C03633=1121.483,37.693,-52.816,179.793,7.035,149.366
C03634=1121.488,37.443,-52.800,179.792,7.030,149.365
C03635=1121.492,37.194,-52.785,179.791,7.026,149.364
C03636=1121.498,36.944,-52.770,179.790,7.022,149.364
C03637=1121.502,36.695,-52.755,179.789,7.018,149.363
C03638=1121.508,36.446,-52.739,179.788,7.014,149.363
C03639=1121.513,36.196,-52.723,179.787,7.010,149.362
C03640=1121.517,35.947,-52.708,179.786,7.006,149.361
C03641=1121.523,35.697,-52.693,179.785,7.002,149.361
C03642=1121.527,35.482,-52.680,179.784,6.997,149.360
C03643=1121.532,35.267,-52.667,179.783,6.994,149.360
C03644=1121.536,35.053,-52.653,179.782,6.991,149.359
C03645=1121.540,34.838,-52.641,179.781,6.987,149.359
C03646=1121.544,34.623,-52.627,179.780,6.983,149.358
C03647=1121.548,34.408,-52.614,179.779,6.979,149.358
C03648=1121.553,34.193,-52.601,179.778,6.976,149.357
C03649=1121.557,33.978,-52.588,179.777,6.973,149.356
C03650=1121.562,33.729,-52.573,179.776,6.968,149.356
C03651=1121.568,33.480,-52.557,179.775,6.964,149.355
C03652=1121.573,33.230,-52.542,179.774,6.960,149.355
C03653=1121.577,32.980,-52.527,179.773,6.955,149.354
C03654=1121.583,32.731,-52.511,179.772,6.951,149.353
C03655=1121.587,32.482,-52.496,179.771,6.947,149.353
C03656=1121.593,32.232,-52.481,179.770,6.942,149.352
C03657=1121.598,31.983,-52.466,179.769,6.938,149.351
C03658=1121.603,31.733,-52.451,179.768,6.934,149.351
C03659=1121.608,31.484,-52.436,179.767,6.929,149.350
C03660=1121.613,31.234,-52.421,179.766,6.925,149.349
C03661=1121.617,30.984,-52.405,179.765,6.921,149.349
C03662=1121.622,30.735,-52.390,179.764,6.916,149.348
C03663=1121.627,30.486,-52.375,179.762,6.912,149.347
C03664=1121.632,30.236,-52.361,179.761,6.908,149.347
C03665=1121.638,29.987,-52.345,179.760,6.904,149.346
C03666=1121.642,29.738,-52.330,179.759,6.899,149.345
C03667=1121.648,29.488,-52.315,179.758,6.895,149.345
C03668=1121.653,29.238,-52.300,179.757,6.891,149.344
C03669=1121.658,28.988,-52.285,179.756,6.886,149.343
C03670=1121.663,28.739,-52.270,179.755,6.882,149.343
C03671=1121.668,28.490,-52.255,179.754,6.878,149.342
C03672=1121.673,28.240,-52.240,179.753,6.873,149.341
C03673=1121.678,27.991,-52.225,179.752,6.869,149.341
C03674=1121.683,27.741,-52.211,179.751,6.864,149.340
C03675=1121.688,27.492,-52.196,179.750,6.860,149.339
C03676=1121.693,27.242,-52.181,179.749,6.856,149.339
C03677=1121.699,26.993,-52.166,179.748,6.851,149.338
C03678=1121.704,26.743,-52.151,179.747,6.847,149.337
C03679=1121.708,26.494,-52.136,179.746,6.843,149.337
C03680=1121.714,26.244,-52.122,179.745,6.838,149.336
C03681=1121.719,25.995,-52.107,179.744,6.834,149.335
C03682=1121.724,25.745,-52.092,179.743,6.829,149.335
C03683=1121.729,25.496,-52.077,179.742,6.825,149.334
C03684=1121.734,25.246,-52.062,179.741,6.821,149.333
C03685=1121.739,24.997,-52.047,179.740,6.816,149.333
C03686=1121.744,24.747,-52.033,179.739,6.812,149.332
C03687=1121.749,24.498,-52.018,179.739,6.807,149.331
C03688=1121.754,24.248,-52.003,179.738,6.803,149.330
C03689=1121.759,23.999,-51.988,179.736,6.799,149.330
C03690=1121.764,23.749,-51.973,179.735,6.794,149.329
C03691=1121.769,23.499,-51.959,179.734,6.790,149.328
C03692=1121.774,23.250,-51.944,179.734,6.785,149.328
C03693=1121.779,23.001,-51.930,179.733,6.781,149.327
C03694=1121.785,22.751,-51.915,179.732,6.777,149.326
C03695=1121.789,22.501,-51.900,179.731,6.772,149.326
C03696=1121.794,22.252,-51.886,179.730,6.768,149.325
C03697=1121.799,22.002,-51.871,179.729,6.763,149.324
C03698=1121.804,21.787,-51.858,179.729,6.760,149.323
C03699=1121.808,21.572,-51.846,179.728,6.756,149.323
C03700=1121.812,21.358,-51.833,179.727,6.752,149.322
C03701=1121.816,21.143,-51.821,179.726,6.749,149.322
C03702=1121.821,20.927,-51.808,179.725,6.745,149.321
C03703=1121.825,20.713,-51.796,179.725,6.741,149.320
C03704=1121.829,20.498,-51.783,179.724,6.737,149.320
C03705=1121.834,20.283,-51.770,179.723,6.733,149.319
C03706=1121.840,20.034,-51.756,179.722,6.729,149.318
C03707=1121.845,19.784,-51.742,179.721,6.725,149.318
C03708=1121.850,19.534,-51.728,179.721,6.720,149.317
C03709=1121.854,19.285,-51.713,179.720,6.716,149.316
C03710=1121.859,19.036,-51.698,179.719,6.711,149.316
C03711=1121.864,18.786,-51.684,179.717,6.706,149.315
C03712=1121.870,18.536,-51.669,179.716,6.701,149.314
C03713=1121.875,18.286,-51.655,179.715,6.697,149.313
C03714=1121.880,18.037,-51.641,179.715,6.692,149.313
C03715=1121.885,17.788,-51.626,179.714,6.688,149.312
C03716=1121.890,17.538,-51.612,179.713,6.683,149.311
C03717=1121.895,17.289,-51.597,179.712,6.679,149.310
C03718=1121.900,17.039,-51.583,179.711,6.675,149.310
C03719=1121.905,16.789,-51.569,179.711,6.670,149.309
C03720=1121.910,16.540,-51.555,179.709,6.666,149.308
C03721=1121.915,16.290,-51.541,179.709,6.661,149.307
C03722=1121.920,16.041,-51.526,179.708,6.657,149.307
C03723=1121.925,15.791,-51.512,179.707,6.652,149.306
C03724=1121.930,15.542,-51.497,179.706,6.648,149.305
C03725=1121.935,15.293,-51.483,179.706,6.643,149.304
C03726=1121.940,15.043,-51.469,179.705,6.639,149.304
C03727=1121.945,14.793,-51.455,179.704,6.634,149.303
C03728=1121.950,14.544,-51.440,179.703,6.630,149.302
C03729=1121.955,14.294,-51.426,179.703,6.625,149.301
C03730=1121.961,14.045,-51.412,179.702,6.621,149.301
C03731=1121.966,13.795,-51.398,179.700,6.615,149.300
C03732=1121.971,13.546,-51.384,179.699,6.611,149.299
C03733=1121.976,13.296,-51.369,179.699,6.606,149.298
C03734=1121.981,13.047,-51.355,179.698,6.602,149.297
C03735=1121.986,12.797,-51.341,179.697,6.597,149.297
C03736=1121.991,12.547,-51.327,179.697,6.592,149.296
C03737=1121.996,12.297,-51.313,179.696,6.588,149.295
C03738=1122.002,12.048,-51.299,179.695,6.583,149.294
C03739=1122.007,11.798,-51.285,179.694,6.579,149.294
C03740=1122.012,11.549,-51.271,179.693,6.574,149.293
C03741=1122.017,11.300,-51.257,179.693,6.569,149.292
C03742=1122.022,11.050,-51.243,179.692,6.565,149.291
C03743=1122.027,10.800,-51.228,179.691,6.560,149.290
C03744=1122.031,10.551,-51.215,179.690,6.555,149.290
C03745=1122.037,10.302,-51.201,179.689,6.551,149.289
C03746=1122.042,10.052,-51.187,179.689,6.546,149.288
C03747=1122.047,9.802,-51.173,179.688,6.542,149.287
C03748=1122.053,9.553,-51.159,179.687,6.537,149.286
C03749=1122.058,9.303,-51.145,179.686,6.532,149.285
C03750=1122.063,9.053,-51.131,179.686,6.527,149.285
C03751=1122.068,8.804,-51.118,179.685,6.523,149.284
C03752=1122.073,8.554,-51.104,179.684,6.518,149.283
C03753=1122.078,8.305,-51.089,179.684,6.514,149.282
C03754=1122.082,8.089,-51.078,179.683,6.509,149.281
C03755=1122.087,7.875,-51.066,179.682,6.506,149.281
C03756=1122.091,7.660,-51.053,179.682,6.502,149.280
C03757=1122.095,7.445,-51.042,179.681,6.498,149.279
C03758=1122.100,7.229,-51.030,179.681,6.494,149.278
C03759=1122.105,7.015,-51.017,179.681,6.490,149.278
C03760=1122.109,6.800,-51.006,179.681,6.487,149.277
C03761=1122.113,6.585,-50.994,179.680,6.482,149.276
C03762=1122.118,6.335,-50.980,179.680,6.477,149.275
C03763=1122.123,6.086,-50.967,179.679,6.474,149.275
C03764=1122.128,5.836,-50.953,179.679,6.469,149.274
C03765=1122.134,5.587,-50.939,179.678,6.464,149.273
C03766=1122.139,5.337,-50.925,179.678,6.459,149.272
C03767=1122.143,5.087,-50.912,179.677,6.455,149.271
C03768=1122.149,4.838,-50.898,179.677,6.451,149.270
C03769=1122.154,4.588,-50.884,179.677,6.446,149.269
C03770=1122.160,4.339,-50.870,179.676,6.442,149.269
C03771=1122.164,4.089,-50.857,179.675,6.437,149.268
C03772=1122.169,3.839,-50.843,179.674,6.432,149.267
C03773=1122.175,3.590,-50.829,179.674,6.428,149.266
C03774=1122.179,3.340,-50.816,179.674,6.424,149.265
C03775=1122.185,3.091,-50.802,179.673,6.419,149.264
C03776=1122.190,2.841,-50.789,179.672,6.415,149.264
C03777=1122.195,2.591,-50.774,179.672,6.410,149.263
C03778=1122.200,2.342,-50.761,179.671,6.405,149.262
C03779=1122.205,2.092,-50.748,179.671,6.400,149.261
C03780=1122.211,1.843,-50.734,179.670,6.397,149.260
C03781=1122.215,1.593,-50.721,179.670,6.392,149.259
C03782=1122.221,1.344,-50.707,179.669,6.387,149.259
C03783=1122.225,1.094,-50.694,179.669,6.383,149.258
C03784=1122.231,0.845,-50.680,179.668,6.378,149.257
C03785=1122.236,0.595,-50.666,179.667,6.374,149.256
C03786=1122.241,0.346,-50.653,179.667,6.370,149.255
C03787=1122.246,0.096,-50.639,179.667,6.365,149.254
C03788=1122.252,-0.153,-50.626,179.666,6.361,149.254
C03789=1122.256,-0.404,-50.613,179.665,6.356,149.253
C03790=1122.262,-0.653,-50.599,179.665,6.351,149.252
C03791=1122.266,-0.903,-50.586,179.664,6.346,149.251
C03792=1122.272,-1.152,-50.573,179.663,6.342,149.250
C03793=1122.276,-1.402,-50.559,179.663,6.338,149.249
C03794=1122.282,-1.651,-50.546,179.663,6.334,149.249
C03795=1122.287,-1.901,-50.531,179.662,6.329,149.248
C03796=1122.292,-2.150,-50.519,179.661,6.324,149.247
C03797=1122.298,-2.401,-50.505,179.661,6.320,149.246
C03798=1122.302,-2.649,-50.492,179.660,6.315,149.245
C03799=1122.308,-2.900,-50.478,179.659,6.311,149.245
C03800=1122.313,-3.149,-50.466,179.659,6.306,149.244
C03801=1122.318,-3.399,-50.451,179.658,6.301,149.243
C03802=1122.323,-3.648,-50.439,179.658,6.297,149.242
C03803=1122.328,-3.898,-50.425,179.657,6.293,149.241
C03804=1122.333,-4.147,-50.412,179.657,6.288,149.240
C03805=1122.338,-4.397,-50.398,179.656,6.284,149.240
C03806=1122.343,-4.647,-50.386,179.655,6.279,149.239
C03807=1122.349,-4.896,-50.373,179.655,6.274,149.238
C03808=1122.353,-5.146,-50.359,179.654,6.270,149.237
C03809=1122.359,-5.395,-50.346,179.653,6.265,149.236
C03810=1122.363,-5.611,-50.334,179.653,6.261,149.236
C03811=1122.368,-5.825,-50.323,179.653,6.258,149.235
C03812=1122.373,-6.041,-50.312,179.652,6.254,149.234
C03813=1122.377,-6.256,-50.300,179.652,6.250,149.234
C03814=1122.382,-6.471,-50.289,179.651,6.246,149.233
C03815=1122.385,-6.686,-50.278,179.650,6.242,149.232
C03816=1122.389,-6.901,-50.266,179.650,6.238,149.231
C03817=1122.394,-7.116,-50.255,179.649,6.234,149.231
C03818=1122.400,-7.367,-50.242,179.648,6.230,149.230
C03819=1122.404,-7.615,-50.229,179.648,6.225,149.229
C03820=1122.410,-7.865,-50.215,179.647,6.220,149.228
C03821=1122.415,-8.115,-50.202,179.646,6.216,149.228
C03822=1122.420,-8.364,-50.190,179.646,6.212,149.227
C03823=1122.426,-8.614,-50.177,179.646,6.207,149.226
C03824=1122.430,-8.864,-50.164,179.645,6.203,149.225
C03825=1122.435,-9.113,-50.151,179.644,6.198,149.224
C03826=1122.441,-9.362,-50.137,179.644,6.193,149.223
C03827=1122.445,-9.612,-50.124,179.643,6.189,149.222
C03828=1122.451,-9.861,-50.112,179.642,6.184,149.222
C03829=1122.456,-10.111,-50.098,179.642,6.179,149.221
C03830=1122.461,-10.361,-50.085,179.641,6.175,149.220
C03831=1122.466,-10.610,-50.073,179.640,6.170,149.219
C03832=1122.472,-10.860,-50.060,179.640,6.166,149.218
C03833=1122.476,-11.110,-50.047,179.639,6.161,149.218
C03834=1122.482,-11.359,-50.034,179.638,6.157,149.217
C03835=1122.487,-11.609,-50.021,179.638,6.152,149.216
C03836=1122.492,-11.859,-50.008,179.637,6.147,149.215
C03837=1122.497,-12.108,-49.995,179.636,6.143,149.214
C03838=1122.502,-12.358,-49.983,179.636,6.138,149.214
C03839=1122.507,-12.608,-49.969,179.635,6.133,149.213
C03840=1122.513,-12.857,-49.956,179.634,6.129,149.212
C03841=1122.518,-13.107,-49.944,179.634,6.124,149.211
C03842=1122.523,-13.356,-49.931,179.633,6.120,149.210
C03843=1122.528,-13.606,-49.918,179.632,6.115,149.210
C03844=1122.533,-13.856,-49.905,179.632,6.110,149.209
C03845=1122.538,-14.105,-49.892,179.631,6.106,149.208
C03846=1122.543,-14.355,-49.880,179.631,6.101,149.207
C03847=1122.549,-14.605,-49.866,179.630,6.097,149.206
C03848=1122.554,-14.854,-49.854,179.629,6.091,149.205
C03849=1122.559,-15.104,-49.842,179.628,6.086,149.204
C03850=1122.564,-15.354,-49.829,179.627,6.082,149.204
C03851=1122.569,-15.603,-49.816,179.627,6.077,149.203
C03852=1122.575,-15.853,-49.803,179.626,6.073,149.202
C03853=1122.580,-16.102,-49.790,179.625,6.068,149.201
C03854=1122.585,-16.351,-49.778,179.625,6.064,149.200
C03855=1122.590,-16.601,-49.765,179.624,6.059,149.200
C03856=1122.595,-16.851,-49.753,179.624,6.054,149.199
C03857=1122.600,-17.101,-49.740,179.623,6.050,149.198
C03858=1122.606,-17.350,-49.727,179.622,6.045,149.197
C03859=1122.611,-17.600,-49.715,179.622,6.040,149.196
C03860=1122.616,-17.850,-49.702,179.621,6.035,149.195
C03861=1122.621,-18.100,-49.690,179.620,6.030,149.195
C03862=1122.626,-18.349,-49.677,179.619,6.026,149.194
C03863=1122.631,-18.598,-49.665,179.619,6.021,149.193
C03864=1122.636,-18.848,-49.652,179.618,6.016,149.192
C03865=1122.641,-19.098,-49.640,179.617,6.012,149.191
C03866=1122.646,-19.313,-49.628,179.617,6.007,149.190
C03867=1122.651,-19.528,-49.618,179.617,6.004,149.190
C03868=1122.655,-19.744,-49.607,179.616,5.999,149.189
C03869=1122.660,-19.959,-49.597,179.615,5.996,149.188
C03870=1122.664,-20.174,-49.585,179.615,5.991,149.188
C03871=1122.668,-20.389,-49.575,179.614,5.987,149.187
C03872=1122.673,-20.605,-49.564,179.613,5.983,149.186
C03873=1122.677,-20.820,-49.554,179.612,5.979,149.186
C03874=1122.683,-21.069,-49.541,179.612,5.974,149.185
C03875=1122.688,-21.319,-49.528,179.612,5.969,149.184
C03876=1122.694,-21.568,-49.516,179.611,5.964,149.183
C03877=1122.699,-21.818,-49.504,179.610,5.959,149.182
C03878=1122.703,-22.068,-49.491,179.609,5.955,149.181
C03879=1122.709,-22.318,-49.479,179.609,5.950,149.180
C03880=1122.714,-22.567,-49.466,179.608,5.945,149.180
C03881=1122.719,-22.817,-49.455,179.608,5.940,149.179
C03882=1122.724,-23.066,-49.442,179.606,5.935,149.178
C03883=1122.730,-23.316,-49.430,179.606,5.930,149.177
C03884=1122.735,-23.566,-49.417,179.605,5.926,149.176
C03885=1122.739,-23.815,-49.405,179.605,5.921,149.175
C03886=1122.745,-24.065,-49.394,179.603,5.916,149.174
C03887=1122.750,-24.314,-49.381,179.603,5.911,149.174
C03888=1122.755,-24.564,-49.369,179.603,5.906,149.173
C03889=1122.760,-24.813,-49.356,179.602,5.901,149.172
C03890=1122.766,-25.063,-49.345,179.601,5.896,149.171
C03891=1122.771,-25.313,-49.333,179.601,5.891,149.170
C03892=1122.776,-25.562,-49.320,179.600,5.886,149.169
C03893=1122.781,-25.813,-49.308,179.598,5.881,149.168
C03894=1122.786,-26.062,-49.295,179.599,5.877,149.167
C03895=1122.792,-26.312,-49.283,179.600,5.872,149.166
C03896=1122.797,-26.561,-49.271,179.601,5.869,149.165
C03897=1122.802,-26.811,-49.259,179.602,5.865,149.164
C03898=1122.807,-27.060,-49.247,179.602,5.860,149.163
C03899=1122.812,-27.310,-49.235,179.603,5.857,149.162
C03900=1122.818,-27.560,-49.223,179.604,5.853,149.161
C03901=1122.823,-27.810,-49.211,179.604,5.848,149.160
C03902=1122.828,-28.060,-49.199,179.605,5.844,149.158
C03903=1122.833,-28.309,-49.186,179.605,5.840,149.158
C03904=1122.838,-28.559,-49.175,179.606,5.836,149.156
C03905=1122.843,-28.808,-49.163,179.607,5.832,149.155
C03906=1122.849,-29.058,-49.150,179.607,5.828,149.154
C03907=1122.854,-29.308,-49.138,179.607,5.823,149.153
C03908=1122.859,-29.558,-49.126,179.607,5.819,149.152
C03909=1122.865,-29.807,-49.114,179.607,5.815,149.151
C03910=1122.869,-30.057,-49.103,179.608,5.811,149.150
C03911=1122.874,-30.306,-49.090,179.608,5.807,149.149
C03912=1122.880,-30.556,-49.078,179.608,5.803,149.148
C03913=1122.885,-30.806,-49.066,179.609,5.799,149.147
C03914=1122.890,-31.055,-49.054,179.608,5.794,149.146
C03915=1122.895,-31.305,-49.042,179.608,5.790,149.146
C03916=1122.900,-31.555,-49.030,179.609,5.786,149.145
C03917=1122.906,-31.805,-49.019,179.608,5.781,149.144
C03918=1122.911,-32.054,-49.006,179.608,5.778,149.143
C03919=1122.916,-32.304,-48.994,179.608,5.773,149.142
C03920=1122.922,-32.553,-48.983,179.608,5.769,149.141
C03921=1122.927,-32.802,-48.971,179.607,5.764,149.140
C03922=1122.931,-33.018,-48.960,179.607,5.761,149.139
C03923=1122.936,-33.233,-48.950,179.607,5.757,149.139
C03924=1122.940,-33.448,-48.940,179.607,5.753,149.138
C03925=1122.945,-33.664,-48.929,179.606,5.749,149.137
C03926=1122.949,-33.879,-48.919,179.606,5.745,149.136
C03927=1122.954,-34.094,-48.909,179.606,5.741,149.136
C03928=1122.959,-34.309,-48.899,179.605,5.738,149.135
C03929=1122.962,-34.525,-48.888,179.605,5.733,149.134
C03930=1122.968,-34.775,-48.876,179.604,5.729,149.133
C03931=1122.973,-35.025,-48.865,179.604,5.724,149.132
C03932=1122.978,-35.273,-48.854,179.603,5.719,149.132
C03933=1122.984,-35.523,-48.842,179.602,5.715,149.131
C03934=1122.989,-35.773,-48.830,179.602,5.710,149.130
C03935=1122.994,-36.023,-48.817,179.601,5.706,149.129
C03936=1122.999,-36.272,-48.806,179.600,5.701,149.128
C03937=1123.005,-36.522,-48.794,179.599,5.695,149.128
C03938=1123.010,-36.772,-48.782,179.598,5.691,149.127
C03939=1123.015,-37.022,-48.771,179.598,5.686,149.126
C03940=1123.020,-37.272,-48.759,179.596,5.681,149.125
C03941=1123.025,-37.521,-48.748,179.596,5.676,149.124
C03942=1123.031,-37.771,-48.736,179.594,5.671,149.124
C03943=1123.036,-38.021,-48.724,179.594,5.666,149.123
C03944=1123.041,-38.270,-48.712,179.592,5.661,149.122
C03945=1123.046,-38.519,-48.700,179.592,5.656,149.121
C03946=1123.051,-38.769,-48.689,179.590,5.651,149.121
C03947=1123.057,-39.018,-48.678,179.589,5.646,149.120
C03948=1123.062,-39.268,-48.666,179.588,5.641,149.119
C03949=1123.067,-39.518,-48.654,179.587,5.636,149.118
C03950=1123.072,-39.768,-48.643,179.586,5.631,149.117
C03951=1123.078,-40.018,-48.631,179.584,5.626,149.117
C03952=1123.083,-40.267,-48.620,179.583,5.620,149.116
C03953=1123.089,-40.517,-48.609,179.582,5.615,149.115
C03954=1123.093,-40.767,-48.597,179.580,5.610,149.115
C03955=1123.099,-41.017,-48.585,179.579,5.603,149.114
C03956=1123.104,-41.266,-48.574,179.577,5.598,149.113
C03957=1123.110,-41.516,-48.563,179.576,5.593,149.112
C03958=1123.114,-41.765,-48.551,179.575,5.587,149.111
C03959=1123.120,-42.015,-48.539,179.572,5.581,149.111
C03960=1123.124,-42.265,-48.528,179.571,5.576,149.110
C03961=1123.130,-42.514,-48.517,179.569,5.570,149.109
C03962=1123.135,-42.764,-48.506,179.568,5.565,149.109
C03963=1123.141,-43.014,-48.494,179.566,5.559,149.108
C03964=1123.146,-43.263,-48.483,179.566,5.554,149.107
C03965=1123.151,-43.513,-48.472,179.566,5.549,149.106
C03966=1123.156,-43.763,-48.460,179.566,5.545,149.105
C03967=1123.161,-44.013,-48.450,179.566,5.540,149.104
C03968=1123.167,-44.262,-48.438,179.567,5.535,149.102
C03969=1123.172,-44.512,-48.427,179.566,5.530,149.101
C03970=1123.177,-44.762,-48.415,179.567,5.526,149.100
C03971=1123.183,-45.011,-48.405,179.567,5.521,149.099
C03972=1123.188,-45.261,-48.393,179.567,5.516,149.098
C03973=1123.193,-45.511,-48.381,179.567,5.512,149.097
C03974=1123.199,-45.760,-48.371,179.567,5.507,149.096
C03975=1123.203,-46.010,-48.360,179.568,5.502,149.095
C03976=1123.209,-46.260,-48.348,179.568,5.497,149.094
C03977=1123.214,-46.509,-48.337,179.567,5.492,149.093
C03978=1123.218,-46.725,-48.327,179.568,5.489,149.092
C03979=1123.223,-46.941,-48.318,179.568,5.485,149.091
C03980=1123.227,-47.156,-48.308,179.568,5.481,149.090
C03981=1123.232,-47.371,-48.299,179.569,5.476,149.089
C03982=1123.237,-47.587,-48.290,179.569,5.472,149.088
C03983=1123.242,-47.802,-48.279,179.569,5.468,149.087
C03984=1123.246,-48.017,-48.270,179.569,5.464,149.086
C03985=1123.251,-48.233,-48.260,179.569,5.460,149.085
C03986=1123.256,-48.482,-48.249,179.569,5.455,149.084
C03987=1123.260,-48.732,-48.238,179.569,5.451,149.083
C03988=1123.267,-48.982,-48.227,179.570,5.446,149.082
C03989=1123.271,-49.231,-48.216,179.570,5.441,149.081
C03990=1123.277,-49.481,-48.206,179.570,5.437,149.080
C03991=1123.282,-49.731,-48.194,179.570,5.432,149.079
C03992=1123.287,-49.981,-48.182,179.571,5.428,149.078
C03993=1123.293,-50.230,-48.172,179.571,5.423,149.077
C03994=1123.297,-50.480,-48.161,179.570,5.418,149.076
C03995=1123.304,-50.730,-48.150,179.571,5.413,149.075
C03996=1123.308,-50.979,-48.139,179.571,5.408,149.073
C03997=1123.313,-51.229,-48.128,179.571,5.404,149.072
C03998=1123.319,-51.478,-48.117,179.571,5.399,149.071
C03999=1123.324,-51.729,-48.106,179.572,5.395,149.070
C04000=1123.330,-51.978,-48.095,179.572,5.390,149.069
C04001=1123.334,-52.227,-48.084,179.572,5.385,149.068
C04002=1123.339,-52.478,-48.073,179.572,5.381,149.067
C04003=1123.345,-52.727,-48.062,179.572,5.376,149.066
C04004=1123.350,-52.977,-48.051,179.573,5.372,149.065
C04005=1123.356,-53.226,-48.040,179.573,5.366,149.064
C04006=1123.361,-53.476,-48.030,179.573,5.361,149.063
C04007=1123.367,-53.726,-48.018,179.573,5.357,149.062
C04008=1123.372,-53.976,-48.008,179.573,5.352,149.061
C04009=1123.377,-54.226,-47.997,179.574,5.348,149.059
C04010=1123.382,-54.475,-47.986,179.573,5.343,149.058
C04011=1123.387,-54.725,-47.976,179.574,5.339,149.057
C04012=1123.392,-54.974,-47.965,179.574,5.334,149.056
C04013=1123.398,-55.225,-47.953,179.574,5.329,149.055
C04014=1123.403,-55.474,-47.943,179.574,5.324,149.054
C04015=1123.408,-55.724,-47.932,179.575,5.319,149.053
C04016=1123.414,-55.973,-47.921,179.575,5.315,149.052
C04017=1123.419,-56.223,-47.910,179.575,5.310,149.051
C04018=1123.424,-56.473,-47.900,179.576,5.306,149.050
C04019=1123.430,-56.723,-47.888,179.575,5.301,149.049
C04020=1123.435,-56.973,-47.878,179.576,5.297,149.048
C04021=1123.440,-57.222,-47.867,179.576,5.292,149.047
C04022=1123.445,-57.472,-47.856,179.576,5.287,149.046
C04023=1123.450,-57.721,-47.846,179.576,5.282,149.044
C04024=1123.455,-57.971,-47.835,179.576,5.278,149.044
C04025=1123.461,-58.221,-47.825,179.577,5.273,149.042
C04026=1123.466,-58.471,-47.814,179.577,5.268,149.041
C04027=1123.471,-58.720,-47.803,179.577,5.264,149.040
C04028=1123.477,-58.970,-47.792,179.577,5.259,149.039
C04029=1123.482,-59.220,-47.782,179.577,5.254,149.038
C04030=1123.487,-59.470,-47.770,179.577,5.250,149.037
C04031=1123.493,-59.719,-47.760,179.577,5.245,149.036
C04032=1123.498,-59.969,-47.750,179.578,5.241,149.035
C04033=1123.503,-60.218,-47.739,179.578,5.236,149.034
C04034=1123.508,-60.434,-47.730,179.577,5.231,149.033
C04035=1123.513,-60.650,-47.721,179.576,5.227,149.032
C04036=1123.516,-60.865,-47.712,179.575,5.222,149.032
C04037=1123.521,-61.081,-47.703,179.575,5.218,149.031
C04038=1123.526,-61.296,-47.694,179.574,5.213,149.030
C04039=1123.530,-61.512,-47.684,179.573,5.209,149.029
C04040=1123.535,-61.727,-47.675,179.573,5.204,149.028
C04041=1123.539,-61.942,-47.666,179.572,5.200,149.028
C04042=1123.545,-62.192,-47.656,179.571,5.194,149.027
C04043=1123.550,-62.442,-47.646,179.571,5.189,149.026
C04044=1123.555,-62.691,-47.635,179.570,5.184,149.025
C04045=1123.560,-62.941,-47.624,179.569,5.179,149.024
C04046=1123.565,-63.191,-47.614,179.568,5.173,149.023
C04047=1123.571,-63.440,-47.604,179.567,5.168,149.022
C04048=1123.576,-63.690,-47.593,179.567,5.163,149.021
C04049=1123.582,-63.940,-47.583,179.566,5.157,149.020
C04050=1123.587,-64.190,-47.572,179.566,5.152,149.019
C04051=1123.592,-64.439,-47.561,179.565,5.147,149.018
C04052=1123.598,-64.689,-47.551,179.564,5.141,149.017
C04053=1123.603,-64.939,-47.541,179.564,5.136,149.016
C04054=1123.608,-65.189,-47.530,179.563,5.131,149.015
C04055=1123.614,-65.438,-47.520,179.563,5.126,149.014
C04056=1123.619,-65.688,-47.510,179.562,5.120,149.013
C04057=1123.624,-65.938,-47.499,179.562,5.115,149.013
C04058=1123.629,-66.187,-47.490,179.561,5.109,149.011
C04059=1123.634,-66.437,-47.479,179.561,5.105,149.011
C04060=1123.640,-66.687,-47.469,179.560,5.099,149.010
C04061=1123.645,-66.936,-47.459,179.560,5.094,149.008
C04062=1123.650,-67.187,-47.448,179.559,5.088,149.008
C04063=1123.656,-67.436,-47.438,179.558,5.084,149.007
C04064=1123.662,-67.686,-47.428,179.558,5.078,149.005
C04065=1123.666,-67.936,-47.418,179.558,5.073,149.005
C04066=1123.671,-68.185,-47.408,179.557,5.067,149.004
C04067=1123.677,-68.435,-47.397,179.557,5.062,149.002
C04068=1123.682,-68.685,-47.387,179.556,5.057,149.002
C04069=1123.688,-68.935,-47.377,179.556,5.052,149.000
C04070=1123.694,-69.185,-47.367,179.555,5.046,148.999
C04071=1123.698,-69.434,-47.357,179.555,5.041,148.998
C04072=1123.703,-69.684,-47.347,179.555,5.036,148.997
C04073=1123.709,-69.934,-47.337,179.554,5.030,148.996
C04074=1123.715,-70.183,-47.326,179.554,5.025,148.995
C04075=1123.719,-70.432,-47.317,179.553,5.019,148.994
C04076=1123.724,-70.683,-47.306,179.553,5.015,148.993
C04077=1123.730,-70.933,-47.297,179.553,5.009,148.992
C04078=1123.736,-71.182,-47.287,179.553,5.003,148.991
C04079=1123.741,-71.432,-47.277,179.552,4.999,148.990
C04080=1123.746,-71.682,-47.266,179.553,4.994,148.989
C04081=1123.751,-71.931,-47.256,179.552,4.988,148.988
C04082=1123.757,-72.182,-47.247,179.552,4.983,148.987
C04083=1123.762,-72.431,-47.237,179.552,4.978,148.986
C04084=1123.768,-72.680,-47.227,179.551,4.972,148.984
C04085=1123.773,-72.931,-47.216,179.551,4.967,148.984
C04086=1123.778,-73.181,-47.207,179.551,4.962,148.982
C04087=1123.784,-73.430,-47.197,179.551,4.956,148.981
C04088=1123.789,-73.680,-47.187,179.550,4.951,148.980
C04089=1123.795,-73.929,-47.177,179.551,4.946,148.979
C04090=1123.799,-74.145,-47.169,179.550,4.941,148.978
C04091=1123.804,-74.361,-47.160,179.550,4.937,148.977
C04092=1123.808,-74.576,-47.152,179.550,4.932,148.976
C04093=1123.813,-74.792,-47.143,179.550,4.927,148.975
C04094=1123.817,-75.007,-47.135,179.550,4.923,148.974
C04095=1123.822,-75.223,-47.126,179.550,4.918,148.973
C04096=1123.826,-75.439,-47.118,179.550,4.914,148.972
C04097=1123.832,-75.654,-47.109,179.550,4.910,148.971
C04098=1123.836,-75.904,-47.100,179.550,4.905,148.970
C04099=1123.842,-76.154,-47.090,179.550,4.899,148.969
C04100=1123.847,-76.403,-47.080,179.550,4.893,148.968
C04101=1123.853,-76.653,-47.071,179.550,4.888,148.967
C04102=1123.858,-76.903,-47.060,179.550,4.884,148.966
C04103=1123.863,-77.152,-47.051,179.550,4.878,148.965
C04104=1123.869,-77.402,-47.041,179.550,4.873,148.964
C04105=1123.874,-77.651,-47.032,179.550,4.868,148.962
C04106=1123.879,-77.902,-47.022,179.550,4.863,148.961
C04107=1123.885,-78.152,-47.012,179.550,4.857,148.960
C04108=1123.890,-78.401,-47.003,179.550,4.852,148.959
C04109=1123.896,-78.651,-46.992,179.550,4.847,148.958
C04110=1123.901,-78.901,-46.984,179.550,4.841,148.957
C04111=1123.906,-79.150,-46.973,179.550,4.836,148.955
C04112=1123.911,-79.400,-46.964,179.551,4.831,148.954
C04113=1123.917,-79.650,-46.954,179.551,4.826,148.953
C04114=1123.922,-79.900,-46.945,179.551,4.821,148.952
C04115=1123.928,-80.149,-46.935,179.551,4.816,148.951
C04116=1123.933,-80.399,-46.926,179.551,4.811,148.950
C04117=1123.938,-80.649,-46.916,179.551,4.805,148.948
C04118=1123.943,-80.899,-46.907,179.552,4.800,148.947
C04119=1123.949,-81.149,-46.897,179.552,4.795,148.946
C04120=1123.954,-81.399,-46.888,179.552,4.790,148.945
C04121=1123.959,-81.648,-46.877,179.552,4.785,148.944
C04122=1123.965,-81.898,-46.869,179.552,4.780,148.943
C04123=1123.970,-82.147,-46.858,179.552,4.774,148.941
C04124=1123.975,-82.397,-46.849,179.553,4.770,148.940
C04125=1123.981,-82.647,-46.840,179.553,4.765,148.939
C04126=1123.986,-82.897,-46.830,179.553,4.760,148.938
C04127=1123.992,-83.147,-46.821,179.554,4.755,148.937
C04128=1123.997,-83.396,-46.811,179.554,4.749,148.935
C04129=1124.002,-83.646,-46.802,179.555,4.744,148.934
C04130=1124.008,-83.896,-46.793,179.555,4.739,148.933
C04131=1124.013,-84.145,-46.783,179.555,4.734,148.932
C04132=1124.019,-84.396,-46.774,179.556,4.729,148.931
C04133=1124.024,-84.645,-46.765,179.556,4.724,148.929
C04134=1124.030,-84.895,-46.755,179.556,4.719,148.928
C04135=1124.035,-85.145,-46.746,179.556,4.714,148.927
C04136=1124.040,-85.395,-46.737,179.557,4.709,148.926
C04137=1124.045,-85.644,-46.727,179.558,4.704,148.924
C04138=1124.051,-85.894,-46.718,179.558,4.699,148.923
C04139=1124.056,-86.144,-46.709,179.558,4.693,148.922
C04140=1124.061,-86.393,-46.699,179.559,4.689,148.921
C04141=1124.067,-86.643,-46.690,179.559,4.684,148.920
C04142=1124.072,-86.893,-46.681,179.559,4.679,148.919
C04143=1124.077,-87.143,-46.671,179.560,4.674,148.917
C04144=1124.083,-87.392,-46.662,179.561,4.669,148.916
C04145=1124.088,-87.643,-46.652,179.561,4.664,148.915
C04146=1124.093,-87.858,-46.644,179.561,4.660,148.914
C04147=1124.097,-88.074,-46.637,179.562,4.655,148.913
C04148=1124.102,-88.289,-46.629,179.562,4.651,148.912
C04149=1124.107,-88.505,-46.620,179.563,4.647,148.911
C04150=1124.111,-88.721,-46.612,179.563,4.643,148.910
C04151=1124.116,-88.936,-46.604,179.564,4.639,148.908
C04152=1124.120,-89.151,-46.597,179.564,4.635,148.907
C04153=1124.125,-89.367,-46.589,179.565,4.630,148.906
C04154=1124.131,-89.617,-46.579,179.565,4.625,148.905
C04155=1124.136,-89.867,-46.570,179.565,4.620,148.904
C04156=1124.141,-90.117,-46.561,179.567,4.615,148.903
C04157=1124.147,-90.367,-46.551,179.567,4.610,148.901
C04158=1124.152,-90.617,-46.542,179.568,4.606,148.900
C04159=1124.157,-90.866,-46.534,179.568,4.601,148.899
C04160=1124.162,-91.116,-46.525,179.569,4.596,148.898
C04161=1124.169,-91.366,-46.516,179.570,4.592,148.896
C04162=1124.173,-91.615,-46.506,179.570,4.586,148.895
C04163=1124.179,-91.865,-46.497,179.571,4.582,148.894
C04164=1124.184,-92.115,-46.488,179.572,4.576,148.893
C04165=1124.190,-92.365,-46.479,179.572,4.572,148.891
C04166=1124.195,-92.615,-46.470,179.573,4.568,148.890
C04167=1124.200,-92.864,-46.461,179.573,4.563,148.889
C04168=1124.206,-93.115,-46.451,179.575,4.558,148.888
C04169=1124.211,-93.365,-46.442,179.575,4.553,148.886
C04170=1124.216,-93.614,-46.433,179.576,4.548,148.885
C04171=1124.222,-93.863,-46.424,179.576,4.544,148.884
C04172=1124.227,-94.113,-46.415,179.578,4.539,148.883
C04173=1124.233,-94.363,-46.406,179.578,4.534,148.881
C04174=1124.238,-94.613,-46.397,179.579,4.530,148.880
C04175=1124.243,-94.863,-46.388,179.579,4.525,148.879
C04176=1124.248,-95.112,-46.379,179.579,4.519,148.878
C04177=1124.254,-95.363,-46.370,179.579,4.514,148.877
C04178=1124.260,-95.612,-46.361,179.580,4.510,148.876
C04179=1124.265,-95.862,-46.352,179.580,4.505,148.875
C04180=1124.270,-96.111,-46.343,179.580,4.500,148.873
C04181=1124.275,-96.361,-46.335,179.580,4.495,148.872
C04182=1124.281,-96.611,-46.326,179.581,4.490,148.871
C04183=1124.286,-96.861,-46.316,179.581,4.485,148.870
C04184=1124.292,-97.111,-46.307,179.581,4.480,148.869
C04185=1124.297,-97.360,-46.299,179.582,4.475,148.867
C04186=1124.303,-97.610,-46.290,179.582,4.470,148.866
C04187=1124.308,-97.860,-46.281,179.583,4.465,148.865
C04188=1124.313,-98.110,-46.272,179.583,4.460,148.864
C04189=1124.318,-98.360,-46.263,179.583,4.455,148.863
C04190=1124.325,-98.609,-46.254,179.583,4.450,148.862
C04191=1124.330,-98.859,-46.245,179.583,4.445,148.861
C04192=1124.335,-99.109,-46.236,179.584,4.441,148.859
C04193=1124.340,-99.359,-46.227,179.584,4.436,148.858
C04194=1124.345,-99.609,-46.218,179.584,4.430,148.857
C04195=1124.351,-99.858,-46.210,179.584,4.425,148.856
C04196=1124.356,-100.108,-46.201,179.585,4.420,148.855
C04197=1124.361,-100.357,-46.192,179.585,4.415,148.853
C04198=1124.367,-100.608,-46.183,179.586,4.411,148.852
C04199=1124.373,-100.858,-46.174,179.586,4.405,148.851
C04200=1124.378,-101.107,-46.166,179.586,4.400,148.850
C04201=1124.384,-101.357,-46.157,179.586,4.395,148.849
C04202=1124.388,-101.573,-46.149,179.587,4.391,148.848
C04203=1124.393,-101.789,-46.142,179.586,4.386,148.847
C04204=1124.397,-102.004,-46.134,179.587,4.382,148.846
C04205=1124.402,-102.220,-46.126,179.587,4.378,148.845
C04206=1124.407,-102.436,-46.119,179.587,4.373,148.844
C04207=1124.411,-102.651,-46.112,179.588,4.369,148.843
C04208=1124.416,-102.867,-46.104,179.588,4.365,148.842
C04209=1124.421,-103.083,-46.097,179.588,4.360,148.841
C04210=1124.426,-103.332,-46.088,179.588,4.355,148.840
C04211=1124.431,-103.582,-46.079,179.588,4.350,148.838
C04212=1124.437,-103.832,-46.071,179.589,4.346,148.837
C04213=1124.442,-104.082,-46.062,179.589,4.341,148.836
C04214=1124.447,-104.332,-46.053,179.589,4.335,148.835
C04215=1124.453,-104.582,-46.044,179.590,4.330,148.834
C04216=1124.458,-104.831,-46.036,179.590,4.325,148.832
C04217=1124.464,-105.081,-46.028,179.590,4.320,148.831
C04218=1124.469,-105.331,-46.019,179.590,4.315,148.830
C04219=1124.475,-105.580,-46.010,179.590,4.310,148.829
C04220=1124.480,-105.830,-46.001,179.590,4.305,148.828
C04221=1124.485,-106.081,-45.993,179.590,4.300,148.827
C04222=1124.491,-106.330,-45.984,179.591,4.294,148.826
C04223=1124.496,-106.580,-45.976,179.591,4.289,148.824
C04224=1124.502,-106.830,-45.968,179.591,4.284,148.823
C04225=1124.506,-107.080,-45.959,179.591,4.279,148.822
C04226=1124.512,-107.329,-45.951,179.592,4.274,148.821
C04227=1124.517,-107.579,-45.943,179.592,4.269,148.820
C04228=1124.523,-107.829,-45.934,179.592,4.263,148.818
C04229=1124.528,-108.078,-45.925,179.592,4.258,148.817
C04230=1124.534,-108.329,-45.917,179.592,4.253,148.816
C04231=1124.539,-108.578,-45.908,179.592,4.248,148.815
C04232=1124.545,-108.828,-45.900,179.593,4.243,148.814
C04233=1124.550,-109.078,-45.891,179.593,4.238,148.813
C04234=1124.555,-109.328,-45.882,179.593,4.233,148.811
C04235=1124.560,-109.577,-45.875,179.593,4.228,148.810
C04236=1124.566,-109.827,-45.866,179.594,4.222,148.809
C04237=1124.572,-110.076,-45.858,179.594,4.217,148.808
C04238=1124.577,-110.327,-45.850,179.594,4.212,148.807
C04239=1124.582,-110.577,-45.841,179.594,4.207,148.805
C04240=1124.588,-110.826,-45.832,179.595,4.202,148.804
C04241=1124.594,-111.076,-45.824,179.595,4.196,148.803
C04242=1124.598,-111.326,-45.816,179.595,4.191,148.802
C04243=1124.604,-111.576,-45.808,179.595,4.186,148.801
C04244=1124.609,-111.826,-45.799,179.596,4.181,148.800
C04245=1124.615,-112.075,-45.791,179.596,4.176,148.798
C04246=1124.620,-112.325,-45.782,179.596,4.171,148.797
C04247=1124.625,-112.575,-45.775,179.596,4.166,148.796
C04248=1124.631,-112.824,-45.766,179.596,4.161,148.795
C04249=1124.636,-113.075,-45.758,179.596,4.155,148.794
C04250=1124.642,-113.324,-45.749,179.596,4.149,148.793
C04251=1124.648,-113.575,-45.741,179.596,4.144,148.791
C04252=1124.653,-113.823,-45.733,179.597,4.139,148.790
C04253=1124.658,-114.074,-45.725,179.597,4.134,148.789
C04254=1124.663,-114.324,-45.716,179.597,4.129,148.788
C04255=1124.669,-114.573,-45.708,179.597,4.124,148.787
C04256=1124.674,-114.824,-45.701,179.598,4.118,148.785
C04257=1124.680,-115.073,-45.692,179.598,4.113,148.784
C04258=1124.684,-115.289,-45.685,179.598,4.108,148.783
C04259=1124.690,-115.505,-45.678,179.598,4.103,148.782
C04260=1124.695,-115.721,-45.671,179.598,4.099,148.781
C04261=1124.698,-115.936,-45.664,179.598,4.095,148.780
C04262=1124.703,-116.152,-45.657,179.599,4.090,148.779
C04263=1124.708,-116.368,-45.650,179.599,4.085,148.778
C04264=1124.713,-116.584,-45.643,179.599,4.081,148.777
C04265=1124.717,-116.799,-45.636,179.599,4.076,148.776
C04266=1124.723,-117.049,-45.628,179.599,4.071,148.775
C04267=1124.729,-117.299,-45.620,179.600,4.066,148.773
C04268=1124.735,-117.549,-45.612,179.599,4.060,148.772
C04269=1124.739,-117.798,-45.604,179.600,4.055,148.771
C04270=1124.745,-118.048,-45.596,179.600,4.050,148.770
C04271=1124.751,-118.299,-45.588,179.600,4.044,148.769
C04272=1124.756,-118.548,-45.580,179.601,4.039,148.767
C04273=1124.761,-118.798,-45.572,179.600,4.033,148.766
C04274=1124.766,-119.047,-45.564,179.601,4.028,148.765
C04275=1124.772,-119.298,-45.556,179.601,4.023,148.764
C04276=1124.778,-119.547,-45.548,179.601,4.018,148.762
C04277=1124.782,-119.797,-45.540,179.601,4.012,148.761
C04278=1124.789,-120.047,-45.532,179.601,4.006,148.760
C04279=1124.794,-120.297,-45.524,179.601,4.001,148.759
C04280=1124.799,-120.546,-45.516,179.602,3.996,148.758
C04281=1124.804,-120.797,-45.508,179.601,3.990,148.756
C04282=1124.810,-121.046,-45.501,179.602,3.985,148.755
C04283=1124.816,-121.296,-45.493,179.602,3.980,148.754
C04284=1124.821,-121.546,-45.485,179.602,3.974,148.753
C04285=1124.826,-121.795,-45.477,179.602,3.969,148.752
C04286=1124.832,-122.046,-45.469,179.603,3.963,148.750
C04287=1124.837,-122.295,-45.461,179.603,3.958,148.749
C04288=1124.843,-122.546,-45.453,179.603,3.952,148.748
C04289=1124.848,-122.795,-45.446,179.603,3.947,148.747
C04290=1124.854,-123.045,-45.438,179.603,3.941,148.745
C04291=1124.859,-123.294,-45.430,179.603,3.935,148.744
C04292=1124.865,-123.544,-45.422,179.603,3.930,148.743
C04293=1124.869,-123.794,-45.414,179.604,3.925,148.742
C04294=1124.875,-124.044,-45.407,179.603,3.919,148.741
C04295=1124.881,-124.294,-45.399,179.604,3.914,148.739
C04296=1124.886,-124.544,-45.391,179.604,3.908,148.738
C04297=1124.892,-124.793,-45.384,179.604,3.902,148.737
C04298=1124.898,-125.043,-45.376,179.604,3.897,148.735
C04299=1124.902,-125.293,-45.369,179.604,3.891,148.734
C04300=1124.908,-125.543,-45.361,179.604,3.886,148.733
C04301=1124.913,-125.793,-45.353,179.605,3.881,148.732
C04302=1124.919,-126.043,-45.345,179.604,3.875,148.731
C04303=1124.925,-126.293,-45.338,179.605,3.869,148.729
C04304=1124.930,-126.543,-45.330,179.605,3.863,148.728
C04305=1124.935,-126.792,-45.323,179.605,3.858,148.727
C04306=1124.941,-127.042,-45.315,179.606,3.853,148.726
C04307=1124.946,-127.292,-45.307,179.605,3.847,148.724
C04308=1124.952,-127.542,-45.300,179.606,3.842,148.723
C04309=1124.958,-127.792,-45.292,179.606,3.835,148.722
C04310=1124.963,-128.041,-45.285,179.606,3.830,148.720
C04311=1124.968,-128.292,-45.277,179.606,3.824,148.719
C04312=1124.974,-128.541,-45.270,179.606,3.819,148.718
C04313=1124.980,-128.791,-45.262,179.606,3.813,148.717
C04314=1124.555,-128.781,-45.288,179.614,3.817,148.715
C04315=1124.551,-128.531,-45.295,179.614,3.823,148.716
C04316=1124.545,-128.282,-45.302,179.613,3.829,148.718
C04317=1124.539,-128.032,-45.310,179.613,3.834,148.719
C04318=1124.535,-127.782,-45.318,179.613,3.840,148.720
C04319=1124.529,-127.532,-45.326,179.613,3.845,148.722
C04320=1124.523,-127.283,-45.333,179.613,3.851,148.723
C04321=1124.518,-127.032,-45.341,179.612,3.857,148.724
C04322=1124.512,-126.783,-45.348,179.613,3.863,148.725
C04323=1124.506,-126.533,-45.356,179.612,3.868,148.727
C04324=1124.502,-126.283,-45.364,179.612,3.873,148.728
C04325=1124.496,-126.033,-45.372,179.612,3.879,148.729
C04326=1124.490,-125.783,-45.379,179.612,3.884,148.730
C04327=1124.485,-125.533,-45.387,179.612,3.891,148.732
C04328=1124.479,-125.284,-45.394,179.611,3.896,148.733
C04329=1124.475,-125.034,-45.402,179.611,3.901,148.734
C04330=1124.469,-124.784,-45.410,179.611,3.907,148.735
C04331=1124.463,-124.534,-45.418,179.611,3.912,148.737
C04332=1124.458,-124.284,-45.426,179.611,3.917,148.738
C04333=1124.452,-124.035,-45.433,179.611,3.923,148.739
C04334=1124.447,-123.784,-45.441,179.611,3.929,148.740
C04335=1124.441,-123.535,-45.449,179.610,3.934,148.742
C04336=1124.436,-123.285,-45.456,179.610,3.940,148.743
C04337=1124.431,-123.035,-45.465,179.610,3.945,148.744
C04338=1124.425,-122.786,-45.472,179.610,3.950,148.745
C04339=1124.420,-122.535,-45.480,179.610,3.956,148.747
C04340=1124.415,-122.286,-45.488,179.610,3.962,148.748
C04341=1124.408,-122.036,-45.495,179.609,3.967,148.749
C04342=1124.403,-121.786,-45.504,179.610,3.973,148.750
C04343=1124.398,-121.537,-45.512,179.609,3.978,148.751
C04344=1124.392,-121.286,-45.520,179.609,3.983,148.753
C04345=1124.387,-121.037,-45.527,179.608,3.989,148.754
C04346=1124.382,-120.786,-45.535,179.609,3.995,148.755
C04347=1124.376,-120.537,-45.544,179.608,4.000,148.756
C04348=1124.371,-120.287,-45.551,179.608,4.005,148.758
C04349=1124.365,-120.037,-45.559,179.608,4.011,148.759
C04350=1124.361,-119.788,-45.567,179.608,4.016,148.760
C04351=1124.355,-119.538,-45.575,179.608,4.021,148.761
C04352=1124.349,-119.288,-45.583,179.607,4.027,148.762
C04353=1124.344,-119.038,-45.591,179.607,4.032,148.764
C04354=1124.338,-118.789,-45.599,179.607,4.038,148.765
C04355=1124.333,-118.538,-45.607,179.607,4.043,148.766
C04356=1124.327,-118.289,-45.615,179.607,4.048,148.767
C04357=1124.322,-118.039,-45.623,179.607,4.053,148.768
C04358=1124.316,-117.789,-45.631,179.607,4.059,148.770
C04359=1124.311,-117.539,-45.639,179.607,4.064,148.771
C04360=1124.305,-117.290,-45.647,179.606,4.070,148.772
C04361=1124.300,-117.040,-45.656,179.606,4.075,148.773
C04362=1124.295,-116.790,-45.664,179.606,4.080,148.774
C04363=1124.290,-116.574,-45.671,179.606,4.085,148.776
C04364=1124.285,-116.359,-45.678,179.605,4.089,148.777
C04365=1124.281,-116.142,-45.685,179.606,4.094,148.778
C04366=1124.276,-115.926,-45.692,179.605,4.099,148.779
C04367=1124.271,-115.711,-45.699,179.605,4.103,148.780
C04368=1124.267,-115.495,-45.706,179.605,4.108,148.781
C04369=1124.262,-115.280,-45.713,179.605,4.112,148.782
C04370=1124.257,-115.064,-45.720,179.605,4.117,148.783
C04371=1124.252,-114.814,-45.729,179.604,4.122,148.784
C04372=1124.246,-114.565,-45.736,179.604,4.127,148.785
C04373=1124.241,-114.314,-45.744,179.604,4.133,148.786
C04374=1124.236,-114.064,-45.753,179.603,4.138,148.788
C04375=1124.230,-113.814,-45.761,179.604,4.144,148.789
C04376=1124.224,-113.565,-45.770,179.604,4.149,148.790
C04377=1124.219,-113.315,-45.777,179.603,4.154,148.791
C04378=1124.214,-113.065,-45.786,179.603,4.159,148.792
C04379=1124.208,-112.816,-45.794,179.603,4.164,148.794
C04380=1124.203,-112.566,-45.803,179.603,4.170,148.795
C04381=1124.198,-112.316,-45.812,179.603,4.174,148.796
C04382=1124.192,-112.066,-45.819,179.603,4.180,148.797
C04383=1124.187,-111.817,-45.828,179.602,4.185,148.798
C04384=1124.181,-111.567,-45.835,179.602,4.190,148.799
C04385=1124.176,-111.317,-45.844,179.602,4.195,148.801
C04386=1124.170,-111.066,-45.853,179.601,4.200,148.802
C04387=1124.165,-110.817,-45.861,179.601,4.205,148.803
C04388=1124.159,-110.567,-45.870,179.601,4.211,148.804
C04389=1124.155,-110.317,-45.878,179.601,4.216,148.805
C04390=1124.149,-110.068,-45.886,179.600,4.221,148.807
C04391=1124.143,-109.818,-45.894,179.600,4.226,148.808
C04392=1124.138,-109.568,-45.903,179.600,4.231,148.809
C04393=1124.133,-109.319,-45.912,179.600,4.237,148.810
C04394=1124.127,-109.068,-45.920,179.600,4.242,148.811
C04395=1124.122,-108.818,-45.929,179.600,4.248,148.813
C04396=1124.116,-108.569,-45.937,179.600,4.253,148.814
C04397=1124.111,-108.319,-45.946,179.599,4.258,148.815
C04398=1124.106,-108.069,-45.954,179.598,4.262,148.816
C04399=1124.100,-107.820,-45.962,179.599,4.267,148.817
C04400=1124.095,-107.570,-45.971,179.599,4.272,148.818
C04401=1124.090,-107.320,-45.979,179.598,4.277,148.820
C04402=1124.084,-107.071,-45.988,179.598,4.283,148.821
C04403=1124.079,-106.820,-45.996,179.598,4.288,148.822
C04404=1124.073,-106.570,-46.005,179.598,4.293,148.823
C04405=1124.068,-106.321,-46.014,179.597,4.298,148.824
C04406=1124.062,-106.071,-46.022,179.597,4.303,148.826
C04407=1124.057,-105.821,-46.031,179.597,4.308,148.827
C04408=1124.051,-105.572,-46.039,179.597,4.314,148.828
C04409=1124.046,-105.322,-46.048,179.596,4.319,148.829
C04410=1124.041,-105.072,-46.057,179.596,4.324,148.830
C04411=1124.035,-104.821,-46.065,179.596,4.329,148.831
C04412=1124.030,-104.572,-46.074,179.596,4.334,148.832
C04413=1124.024,-104.322,-46.083,179.596,4.339,148.834
C04414=1124.019,-104.073,-46.092,179.596,4.344,148.835
C04415=1124.014,-103.823,-46.100,179.595,4.349,148.836
C04416=1124.008,-103.573,-46.108,179.595,4.354,148.837
C04417=1124.003,-103.323,-46.117,179.594,4.359,148.838
C04418=1123.998,-103.073,-46.126,179.594,4.364,148.840
C04419=1123.993,-102.858,-46.134,179.594,4.369,148.841
C04420=1123.988,-102.642,-46.141,179.594,4.373,148.841
C04421=1123.984,-102.427,-46.149,179.593,4.377,148.843
C04422=1123.979,-102.211,-46.156,179.594,4.382,148.844
C04423=1123.974,-101.995,-46.163,179.593,4.386,148.845
C04424=1123.970,-101.779,-46.171,179.593,4.390,148.846
C04425=1123.965,-101.564,-46.179,179.593,4.395,148.847
C04426=1123.961,-101.348,-46.186,179.593,4.399,148.848
C04427=1123.956,-101.098,-46.195,179.592,4.404,148.849
C04428=1123.950,-100.848,-46.204,179.592,4.409,148.850
C04429=1123.944,-100.599,-46.213,179.592,4.414,148.851
C04430=1123.939,-100.349,-46.222,179.592,4.419,148.852
C04431=1123.934,-100.099,-46.231,179.591,4.424,148.853
C04432=1123.928,-99.849,-46.240,179.591,4.429,148.855
C04433=1123.923,-99.599,-46.249,179.591,4.434,148.856
C04434=1123.917,-99.350,-46.257,179.591,4.439,148.857
C04435=1123.912,-99.100,-46.266,179.590,4.444,148.858
C04436=1123.907,-98.850,-46.275,179.590,4.449,148.859
C04437=1123.901,-98.600,-46.285,179.589,4.454,148.861
C04438=1123.896,-98.350,-46.293,179.589,4.459,148.862
C04439=1123.890,-98.101,-46.302,179.589,4.464,148.863
C04440=1123.885,-97.851,-46.311,179.589,4.469,148.864
C04441=1123.880,-97.601,-46.320,179.588,4.473,148.865
C04442=1123.875,-97.352,-46.329,179.588,4.479,148.866
C04443=1123.869,-97.101,-46.338,179.588,4.484,148.867
C04444=1123.864,-96.852,-46.347,179.588,4.489,148.869
C04445=1123.858,-96.602,-46.356,179.588,4.494,148.870
C04446=1123.853,-96.353,-46.365,179.587,4.498,148.871
C04447=1123.848,-96.103,-46.373,179.587,4.504,148.872
C04448=1123.842,-95.853,-46.382,179.586,4.509,148.873
C04449=1123.837,-95.603,-46.392,179.586,4.514,148.874
C04450=1123.831,-95.353,-46.401,179.585,4.518,148.876
C04451=1123.826,-95.103,-46.410,179.585,4.524,148.877
C04452=1123.821,-94.853,-46.419,179.586,4.528,148.878
C04453=1123.815,-94.604,-46.428,179.585,4.533,148.879
C04454=1123.809,-94.354,-46.437,179.585,4.538,148.880
C04455=1123.804,-94.104,-46.445,179.583,4.543,148.882
C04456=1123.799,-93.855,-46.455,179.583,4.548,148.883
C04457=1123.793,-93.605,-46.465,179.582,4.552,148.884
C04458=1123.788,-93.355,-46.473,179.581,4.556,148.885
C04459=1123.783,-93.105,-46.482,179.581,4.562,148.887
C04460=1123.778,-92.855,-46.491,179.580,4.566,148.888
C04461=1123.772,-92.605,-46.501,179.580,4.572,148.889
C04462=1123.766,-92.356,-46.509,179.579,4.576,148.890
C04463=1123.761,-92.107,-46.519,179.578,4.581,148.892
C04464=1123.756,-91.857,-46.528,179.577,4.586,148.893
C04465=1123.750,-91.607,-46.537,179.577,4.590,148.894
C04466=1123.745,-91.357,-46.546,179.576,4.595,148.895
C04467=1123.740,-91.107,-46.555,179.575,4.600,148.897
C04468=1123.735,-90.858,-46.565,179.575,4.605,148.898
C04469=1123.729,-90.607,-46.574,179.574,4.610,148.899
C04470=1123.724,-90.358,-46.583,179.573,4.614,148.900
C04471=1123.719,-90.108,-46.592,179.573,4.619,148.902
C04472=1123.713,-89.858,-46.601,179.573,4.625,148.903
C04473=1123.708,-89.608,-46.611,179.572,4.629,148.904
C04474=1123.703,-89.358,-46.620,179.572,4.634,148.905
C04475=1123.697,-89.143,-46.628,179.571,4.638,148.906
C04476=1123.693,-88.927,-46.636,179.571,4.642,148.907
C04477=1123.689,-88.711,-46.644,179.570,4.647,148.908
C04478=1123.684,-88.496,-46.652,179.569,4.651,148.909
C04479=1123.679,-88.280,-46.660,179.569,4.655,148.910
C04480=1123.674,-88.065,-46.668,179.568,4.659,148.911
C04481=1123.670,-87.849,-46.676,179.568,4.663,148.913
C04482=1123.666,-87.634,-46.684,179.567,4.667,148.914
C04483=1123.660,-87.383,-46.693,179.567,4.673,148.915
C04484=1123.655,-87.134,-46.703,179.567,4.678,148.916
C04485=1123.650,-86.884,-46.712,179.566,4.682,148.917
C04486=1123.644,-86.634,-46.721,179.566,4.688,148.918
C04487=1123.639,-86.384,-46.730,179.565,4.693,148.920
C04488=1123.633,-86.135,-46.741,179.565,4.698,148.921
C04489=1123.628,-85.885,-46.749,179.564,4.702,148.922
C04490=1123.623,-85.635,-46.758,179.564,4.708,148.923
C04491=1123.617,-85.385,-46.769,179.564,4.713,148.925
C04492=1123.612,-85.136,-46.777,179.563,4.718,148.926
C04493=1123.607,-84.886,-46.788,179.563,4.723,148.927
C04494=1123.602,-84.636,-46.797,179.562,4.728,148.928
C04495=1123.596,-84.386,-46.805,179.562,4.733,148.929
C04496=1123.591,-84.137,-46.816,179.562,4.738,148.930
C04497=1123.586,-83.887,-46.825,179.562,4.743,148.932
C04498=1123.580,-83.637,-46.834,179.561,4.748,148.933
C04499=1123.575,-83.388,-46.844,179.560,4.753,148.934
C04500=1123.569,-83.137,-46.853,179.560,4.758,148.935
C04501=1123.564,-82.888,-46.863,179.560,4.763,148.937
C04502=1123.559,-82.638,-46.872,179.560,4.769,148.938
C04503=1123.553,-82.389,-46.882,179.560,4.774,148.939
C04504=1123.548,-82.139,-46.891,179.560,4.779,148.940
C04505=1123.542,-81.889,-46.900,179.559,4.784,148.941
C04506=1123.537,-81.640,-46.910,179.559,4.788,148.942
C04507=1123.531,-81.389,-46.919,179.559,4.794,148.944
C04508=1123.527,-81.140,-46.929,179.558,4.799,148.945
C04509=1123.521,-80.890,-46.938,179.558,4.804,148.946
C04510=1123.516,-80.640,-46.948,179.558,4.809,148.947
C04511=1123.511,-80.390,-46.958,179.558,4.814,148.948
C04512=1123.506,-80.141,-46.968,179.558,4.819,148.949
C04513=1123.500,-79.891,-46.977,179.558,4.825,148.951
C04514=1123.495,-79.641,-46.987,179.557,4.830,148.952
C04515=1123.489,-79.391,-46.996,179.557,4.835,148.953
C04516=1123.483,-79.142,-47.006,179.557,4.840,148.954
C04517=1123.479,-78.892,-47.016,179.557,4.845,148.955
C04518=1123.473,-78.642,-47.025,179.557,4.850,148.956
C04519=1123.468,-78.393,-47.035,179.557,4.855,148.958
C04520=1123.462,-78.143,-47.045,179.557,4.861,148.959
C04521=1123.458,-77.893,-47.055,179.557,4.867,148.960
C04522=1123.452,-77.643,-47.064,179.557,4.872,148.961
C04523=1123.446,-77.393,-47.074,179.557,4.877,148.962
C04524=1123.441,-77.144,-47.084,179.556,4.882,148.963
C04525=1123.435,-76.894,-47.093,179.556,4.887,148.965
C04526=1123.430,-76.644,-47.104,179.556,4.892,148.966
C04527=1123.425,-76.395,-47.113,179.556,4.897,148.967
C04528=1123.420,-76.144,-47.123,179.557,4.903,148.968
C04529=1123.415,-75.895,-47.133,179.557,4.908,148.969
C04530=1123.409,-75.645,-47.142,179.557,4.913,148.970
C04531=1123.404,-75.429,-47.151,179.557,4.918,148.971
C04532=1123.399,-75.214,-47.159,179.557,4.922,148.972
C04533=1123.395,-74.999,-47.168,179.557,4.927,148.973
C04534=1123.390,-74.783,-47.176,179.556,4.931,148.974
C04535=1123.386,-74.567,-47.186,179.557,4.936,148.975
C04536=1123.381,-74.352,-47.193,179.557,4.941,148.976
C04537=1123.376,-74.137,-47.202,179.557,4.945,148.977
C04538=1123.372,-73.921,-47.210,179.557,4.950,148.978
C04539=1123.367,-73.671,-47.221,179.557,4.955,148.979
C04540=1123.361,-73.421,-47.230,179.557,4.961,148.980
C04541=1123.356,-73.172,-47.240,179.558,4.965,148.981
C04542=1123.351,-72.922,-47.250,179.558,4.971,148.982
C04543=1123.345,-72.672,-47.261,179.558,4.976,148.983
C04544=1123.340,-72.423,-47.270,179.559,4.981,148.984
C04545=1123.334,-72.173,-47.280,179.558,4.987,148.986
C04546=1123.329,-71.923,-47.290,179.558,4.992,148.987
C04547=1123.324,-71.673,-47.300,179.559,4.997,148.988
C04548=1123.319,-71.424,-47.310,179.559,5.002,148.989
C04549=1123.313,-71.174,-47.320,179.559,5.008,148.990
C04550=1123.308,-70.923,-47.330,179.560,5.013,148.991
C04551=1123.302,-70.674,-47.340,179.560,5.018,148.992
C04552=1123.297,-70.424,-47.351,179.560,5.023,148.993
C04553=1123.292,-70.175,-47.360,179.561,5.029,148.994
C04554=1123.287,-69.925,-47.371,179.561,5.034,148.995
C04555=1123.281,-69.675,-47.381,179.561,5.040,148.996
C04556=1123.276,-69.426,-47.391,179.562,5.044,148.997
C04557=1123.270,-69.176,-47.401,179.562,5.050,148.998
C04558=1123.266,-68.926,-47.411,179.563,5.055,148.999
C04559=1123.260,-68.677,-47.422,179.562,5.060,149.000
C04560=1123.254,-68.427,-47.431,179.563,5.066,149.001
C04561=1123.249,-68.176,-47.442,179.563,5.071,149.002
C04562=1123.244,-67.927,-47.452,179.564,5.077,149.003
C04563=1123.238,-67.677,-47.462,179.564,5.082,149.004
C04564=1123.234,-67.427,-47.472,179.565,5.087,149.005
C04565=1123.228,-67.178,-47.482,179.565,5.092,149.006
C04566=1123.223,-66.928,-47.492,179.565,5.097,149.007
C04567=1123.218,-66.678,-47.503,179.566,5.103,149.008
C04568=1123.212,-66.428,-47.513,179.567,5.108,149.009
C04569=1123.207,-66.179,-47.523,179.567,5.114,149.010
C04570=1123.202,-65.929,-47.535,179.568,5.118,149.011
C04571=1123.196,-65.680,-47.545,179.569,5.124,149.012
C04572=1123.191,-65.430,-47.555,179.568,5.129,149.013
C04573=1123.186,-65.180,-47.565,179.569,5.135,149.014
C04574=1123.181,-64.931,-47.575,179.570,5.140,149.015
C04575=1123.175,-64.681,-47.586,179.571,5.145,149.016
C04576=1123.170,-64.431,-47.596,179.572,5.151,149.017
C04577=1123.165,-64.181,-47.606,179.572,5.156,149.018
C04578=1123.160,-63.931,-47.617,179.573,5.161,149.019
C04579=1123.154,-63.682,-47.627,179.573,5.166,149.020
C04580=1123.149,-63.433,-47.638,179.574,5.172,149.021
C04581=1123.144,-63.182,-47.649,179.575,5.177,149.022
C04582=1123.138,-62.933,-47.659,179.575,5.182,149.023
C04583=1123.133,-62.683,-47.669,179.576,5.187,149.024
C04584=1123.128,-62.433,-47.680,179.577,5.192,149.025
C04585=1123.123,-62.183,-47.691,179.578,5.198,149.026
C04586=1123.117,-61.934,-47.701,179.579,5.203,149.026
C04587=1123.113,-61.718,-47.710,179.579,5.208,149.027
C04588=1123.108,-61.503,-47.720,179.580,5.212,149.028
C04589=1123.103,-61.287,-47.729,179.580,5.217,149.029
C04590=1123.099,-61.072,-47.738,179.581,5.222,149.030
C04591=1123.095,-60.857,-47.747,179.582,5.226,149.030
C04592=1123.090,-60.641,-47.756,179.583,5.231,149.031
C04593=1123.086,-60.426,-47.766,179.583,5.235,149.032
C04594=1123.081,-60.210,-47.775,179.584,5.240,149.033
C04595=1123.075,-59.961,-47.785,179.584,5.244,149.034
C04596=1123.070,-59.711,-47.796,179.583,5.249,149.035
C04597=1123.065,-59.462,-47.807,179.583,5.253,149.036
C04598=1123.060,-59.211,-47.817,179.583,5.258,149.037
C04599=1123.054,-58.962,-47.827,179.583,5.263,149.038
C04600=1123.050,-58.712,-47.839,179.583,5.267,149.039
C04601=1123.044,-58.463,-47.849,179.583,5.272,149.040
C04602=1123.039,-58.212,-47.859,179.582,5.277,149.041
C04603=1123.033,-57.963,-47.871,179.582,5.281,149.042
C04604=1123.028,-57.713,-47.881,179.582,5.286,149.043
C04605=1123.022,-57.463,-47.892,179.582,5.291,149.044
C04606=1123.018,-57.214,-47.903,179.581,5.295,149.046
C04607=1123.012,-56.964,-47.913,179.581,5.300,149.047
C04608=1123.008,-56.715,-47.924,179.582,5.305,149.048
C04609=1123.002,-56.465,-47.935,179.581,5.309,149.049
C04610=1122.996,-56.214,-47.946,179.581,5.314,149.050
C04611=1122.991,-55.965,-47.957,179.581,5.318,149.051
C04612=1122.986,-55.715,-47.967,179.581,5.323,149.052
C04613=1122.981,-55.466,-47.979,179.580,5.328,149.053
C04614=1122.976,-55.216,-47.989,179.580,5.332,149.054
C04615=1122.971,-54.967,-48.000,179.580,5.338,149.055
C04616=1122.965,-54.717,-48.011,179.580,5.342,149.056
C04617=1122.960,-54.467,-48.022,179.580,5.347,149.057
C04618=1122.955,-54.217,-48.033,179.579,5.351,149.058
C04619=1122.950,-53.968,-48.044,179.579,5.356,149.060
C04620=1122.945,-53.718,-48.054,179.579,5.360,149.060
C04621=1122.939,-53.468,-48.066,179.579,5.365,149.062
C04622=1122.934,-53.218,-48.076,179.579,5.370,149.063
C04623=1122.928,-52.969,-48.087,179.579,5.374,149.064
C04624=1122.923,-52.719,-48.098,179.579,5.380,149.065
C04625=1122.918,-52.469,-48.110,179.578,5.384,149.066
C04626=1122.912,-52.219,-48.120,179.578,5.389,149.067
C04627=1122.908,-51.970,-48.131,179.578,5.393,149.068
C04628=1122.902,-51.720,-48.141,179.578,5.398,149.069
C04629=1122.897,-51.470,-48.153,179.578,5.403,149.070
C04630=1122.892,-51.221,-48.165,179.577,5.407,149.071
C04631=1122.886,-50.971,-48.175,179.577,5.412,149.072
C04632=1122.881,-50.721,-48.187,179.577,5.417,149.074
C04633=1122.875,-50.472,-48.197,179.577,5.421,149.074
C04634=1122.871,-50.222,-48.208,179.577,5.427,149.076
C04635=1122.866,-49.972,-48.219,179.576,5.431,149.077
C04636=1122.859,-49.723,-48.230,179.577,5.436,149.078
C04637=1122.855,-49.473,-48.242,179.576,5.440,149.079
C04638=1122.850,-49.223,-48.252,179.576,5.445,149.080
C04639=1122.844,-48.974,-48.264,179.575,5.449,149.081
C04640=1122.839,-48.724,-48.275,179.576,5.454,149.082
C04641=1122.834,-48.474,-48.286,179.576,5.459,149.083
C04642=1122.828,-48.224,-48.297,179.575,5.464,149.084
C04643=1122.823,-48.009,-48.306,179.575,5.468,149.085
C04644=1122.819,-47.794,-48.316,179.575,5.472,149.086
C04645=1122.814,-47.579,-48.326,179.574,5.476,149.087
C04646=1122.810,-47.363,-48.335,179.575,5.480,149.088
C04647=1122.806,-47.148,-48.345,179.575,5.484,149.089
C04648=1122.801,-46.932,-48.355,179.574,5.488,149.090
C04649=1122.797,-46.717,-48.364,179.574,5.492,149.091
C04650=1122.792,-46.502,-48.374,179.574,5.496,149.092
C04651=1122.787,-46.252,-48.386,179.574,5.501,149.093
C04652=1122.781,-46.002,-48.396,179.573,5.506,149.094
C04653=1122.777,-45.753,-48.407,179.574,5.510,149.095
C04654=1122.771,-45.503,-48.419,179.573,5.515,149.096
C04655=1122.766,-45.254,-48.430,179.573,5.520,149.097
C04656=1122.760,-45.003,-48.441,179.573,5.525,149.098
C04657=1122.756,-44.753,-48.453,179.573,5.529,149.099
C04658=1122.750,-44.505,-48.464,179.573,5.534,149.100
C04659=1122.745,-44.255,-48.475,179.572,5.538,149.101
C04660=1122.740,-44.004,-48.486,179.572,5.544,149.103
C04661=1122.734,-43.754,-48.498,179.572,5.547,149.103
C04662=1122.729,-43.506,-48.509,179.572,5.553,149.105
C04663=1122.724,-43.256,-48.521,179.572,5.558,149.106
C04664=1122.719,-43.006,-48.532,179.572,5.563,149.107
C04665=1122.713,-42.756,-48.543,179.573,5.568,149.108
C04666=1122.708,-42.506,-48.554,179.575,5.574,149.108
C04667=1122.703,-42.257,-48.565,179.577,5.579,149.109
C04668=1122.698,-42.007,-48.577,179.579,5.586,149.110
C04669=1122.693,-41.758,-48.588,179.580,5.591,149.110
C04670=1122.687,-41.508,-48.600,179.582,5.596,149.111
C04671=1122.682,-41.258,-48.611,179.583,5.602,149.112
C04672=1122.677,-41.009,-48.623,179.585,5.607,149.113
C04673=1122.672,-40.759,-48.635,179.586,5.613,149.114
C04674=1122.666,-40.510,-48.646,179.587,5.618,149.114
C04675=1122.661,-40.260,-48.658,179.589,5.623,149.115
C04676=1122.656,-40.010,-48.669,179.590,5.629,149.116
C04677=1122.651,-39.760,-48.681,179.591,5.634,149.116
C04678=1122.646,-39.511,-48.692,179.593,5.639,149.117
C04679=1122.640,-39.261,-48.704,179.594,5.645,149.118
C04680=1122.635,-39.011,-48.716,179.595,5.649,149.119
C04681=1122.630,-38.762,-48.727,179.596,5.655,149.120
C04682=1122.624,-38.512,-48.739,179.598,5.660,149.120
C04683=1122.620,-38.262,-48.750,179.598,5.664,149.121
C04684=1122.614,-38.012,-48.762,179.600,5.670,149.122
C04685=1122.608,-37.763,-48.774,179.600,5.674,149.123
C04686=1122.604,-37.513,-48.785,179.602,5.680,149.123
C04687=1122.598,-37.263,-48.797,179.602,5.684,149.124
C04688=1122.593,-37.013,-48.809,179.603,5.689,149.125
C04689=1122.588,-36.764,-48.820,179.604,5.694,149.126
C04690=1122.583,-36.515,-48.833,179.605,5.699,149.127
C04691=1122.577,-36.265,-48.844,179.606,5.704,149.127
C04692=1122.572,-36.015,-48.856,179.606,5.709,149.128
C04693=1122.567,-35.765,-48.868,179.607,5.713,149.129
C04694=1122.561,-35.516,-48.879,179.608,5.718,149.130
C04695=1122.556,-35.266,-48.891,179.608,5.723,149.131
C04696=1122.552,-35.017,-48.903,179.609,5.727,149.131
C04697=1122.546,-34.767,-48.915,179.610,5.732,149.132
C04698=1122.541,-34.517,-48.927,179.610,5.736,149.133
C04699=1122.536,-34.302,-48.937,179.610,5.740,149.134
C04700=1122.532,-34.086,-48.948,179.611,5.744,149.135
C04701=1122.527,-33.871,-48.958,179.612,5.748,149.135
C04702=1122.523,-33.657,-48.968,179.612,5.752,149.136
C04703=1122.518,-33.440,-48.978,179.612,5.755,149.137
C04704=1122.514,-33.225,-48.988,179.613,5.760,149.138
C04705=1122.509,-33.010,-48.999,179.613,5.764,149.138
C04706=1122.505,-32.795,-49.009,179.613,5.767,149.139
C04707=1122.499,-32.545,-49.021,179.613,5.771,149.140
C04708=1122.494,-32.296,-49.033,179.613,5.776,149.141
C04709=1122.489,-32.046,-49.044,179.614,5.781,149.142
C04710=1122.484,-31.796,-49.056,179.614,5.785,149.143
C04711=1122.479,-31.547,-49.069,179.614,5.789,149.144
C04712=1122.473,-31.297,-49.081,179.614,5.793,149.145
C04713=1122.468,-31.047,-49.093,179.614,5.797,149.145
C04714=1122.464,-30.798,-49.105,179.613,5.802,149.147
C04715=1122.458,-30.548,-49.117,179.614,5.806,149.148
C04716=1122.453,-30.298,-49.129,179.614,5.810,149.148
C04717=1122.448,-30.049,-49.141,179.613,5.814,149.149
C04718=1122.442,-29.799,-49.153,179.613,5.819,149.150
C04719=1122.437,-29.550,-49.166,179.613,5.823,149.151
C04720=1122.432,-29.300,-49.177,179.612,5.826,149.152
C04721=1122.427,-29.050,-49.189,179.612,5.831,149.153
C04722=1122.422,-28.801,-49.201,179.612,5.835,149.154
C04723=1122.416,-28.551,-49.213,179.611,5.839,149.155
C04724=1122.411,-28.301,-49.226,179.610,5.843,149.157
C04725=1122.406,-28.052,-49.238,179.610,5.847,149.157
C04726=1122.400,-27.802,-49.250,179.610,5.852,149.159
C04727=1122.396,-27.553,-49.262,179.609,5.856,149.160
C04728=1122.391,-27.303,-49.274,179.609,5.860,149.161
C04729=1122.385,-27.053,-49.286,179.608,5.864,149.162
C04730=1122.380,-26.803,-49.298,179.607,5.868,149.163
C04731=1122.375,-26.553,-49.311,179.606,5.872,149.164
C04732=1122.370,-26.303,-49.323,179.605,5.876,149.165
C04733=1122.365,-26.054,-49.335,179.605,5.880,149.166
C04734=1122.359,-25.804,-49.347,179.605,5.885,149.167
C04735=1122.354,-25.555,-49.360,179.606,5.890,149.168
C04736=1122.350,-25.305,-49.371,179.606,5.894,149.169
C04737=1122.345,-25.056,-49.384,179.607,5.899,149.170
C04738=1122.339,-24.806,-49.396,179.608,5.905,149.171
C04739=1122.334,-24.557,-49.408,179.608,5.909,149.172
C04740=1122.329,-24.307,-49.420,179.609,5.914,149.173
C04741=1122.323,-24.057,-49.433,179.609,5.919,149.173
C04742=1122.318,-23.807,-49.445,179.610,5.924,149.174
C04743=1122.313,-23.558,-49.457,179.611,5.929,149.175
C04744=1122.307,-23.308,-49.469,179.612,5.933,149.176
C04745=1122.302,-23.059,-49.482,179.612,5.938,149.177
C04746=1122.297,-22.809,-49.494,179.613,5.944,149.178
C04747=1122.292,-22.559,-49.507,179.614,5.948,149.179
C04748=1122.287,-22.310,-49.519,179.614,5.953,149.180
C04749=1122.282,-22.060,-49.531,179.615,5.957,149.180
C04750=1122.277,-21.810,-49.544,179.616,5.962,149.181
C04751=1122.271,-21.560,-49.556,179.617,5.968,149.182
C04752=1122.266,-21.311,-49.568,179.617,5.972,149.183
C04753=1122.261,-21.062,-49.581,179.618,5.977,149.184
C04754=1122.256,-20.812,-49.593,179.618,5.982,149.185
C04755=1122.251,-20.597,-49.604,179.619,5.986,149.185
C04756=1122.246,-20.381,-49.615,179.619,5.990,149.186
C04757=1122.243,-20.166,-49.625,179.620,5.994,149.187
C04758=1122.238,-19.951,-49.637,179.621,5.999,149.188
C04759=1122.233,-19.736,-49.647,179.621,6.002,149.188
C04760=1122.229,-19.521,-49.658,179.622,6.007,149.189
C04761=1122.224,-19.306,-49.669,179.623,6.010,149.190
C04762=1122.220,-19.090,-49.680,179.623,6.015,149.190
C04763=1122.215,-18.841,-49.693,179.624,6.019,149.191
C04764=1122.209,-18.591,-49.704,179.624,6.024,149.192
C04765=1122.204,-18.342,-49.717,179.625,6.029,149.193
C04766=1122.200,-18.092,-49.730,179.625,6.034,149.194
C04767=1122.194,-17.842,-49.743,179.626,6.038,149.194
C04768=1122.189,-17.593,-49.755,179.628,6.043,149.195
C04769=1122.184,-17.343,-49.767,179.628,6.048,149.196
C04770=1122.178,-17.093,-49.780,179.629,6.053,149.197
C04771=1122.174,-16.843,-49.793,179.629,6.057,149.198
C04772=1122.168,-16.594,-49.806,179.630,6.062,149.199
C04773=1122.163,-16.345,-49.818,179.630,6.067,149.200
C04774=1122.158,-16.095,-49.831,179.631,6.071,149.200
C04775=1122.153,-15.845,-49.843,179.632,6.076,149.201
C04776=1122.147,-15.595,-49.856,179.632,6.081,149.202
C04777=1122.142,-15.346,-49.869,179.633,6.085,149.203
C04778=1122.137,-15.096,-49.882,179.634,6.090,149.204
C04779=1122.132,-14.847,-49.894,179.634,6.094,149.204
C04780=1122.127,-14.597,-49.908,179.635,6.099,149.205
C04781=1122.122,-14.347,-49.920,179.635,6.104,149.206
C04782=1122.117,-14.098,-49.933,179.636,6.108,149.207
C04783=1122.111,-13.849,-49.946,179.637,6.114,149.208
C04784=1122.107,-13.599,-49.959,179.638,6.118,149.209
C04785=1122.101,-13.349,-49.972,179.639,6.123,149.209
C04786=1122.096,-13.100,-49.984,179.639,6.128,149.210
C04787=1122.091,-12.850,-49.997,179.640,6.132,149.211
C04788=1122.086,-12.600,-50.011,179.641,6.137,149.212
C04789=1122.080,-12.351,-50.023,179.641,6.141,149.213
C04790=1122.076,-12.101,-50.036,179.642,6.146,149.214
C04791=1122.071,-11.852,-50.049,179.642,6.151,149.214
C04792=1122.065,-11.602,-50.062,179.643,6.155,149.215
C04793=1122.060,-11.353,-50.075,179.644,6.160,149.216
C04794=1122.055,-11.103,-50.087,179.644,6.165,149.217
C04795=1122.049,-10.853,-50.101,179.645,6.169,149.218
C04796=1122.044,-10.604,-50.113,179.646,6.174,149.218
C04797=1122.040,-10.354,-50.126,179.646,6.178,149.219
C04798=1122.034,-10.104,-50.139,179.647,6.183,149.220
C04799=1122.029,-9.854,-50.152,179.648,6.187,149.221
C04800=1122.024,-9.605,-50.165,179.648,6.192,149.222
C04801=1122.018,-9.355,-50.178,179.649,6.196,149.222
C04802=1122.014,-9.106,-50.192,179.649,6.200,149.223
C04803=1122.009,-8.856,-50.204,179.650,6.205,149.224
C04804=1122.003,-8.607,-50.218,179.651,6.210,149.225
C04805=1121.999,-8.357,-50.231,179.651,6.214,149.226
C04806=1121.993,-8.107,-50.244,179.652,6.219,149.227
C04807=1121.988,-7.857,-50.257,179.653,6.223,149.227
C04808=1121.983,-7.608,-50.269,179.653,6.228,149.228
C04809=1121.978,-7.359,-50.283,179.654,6.233,149.229
C04810=1121.973,-7.109,-50.296,179.655,6.237,149.230
C04811=1121.968,-6.894,-50.308,179.655,6.241,149.231
C04812=1121.964,-6.678,-50.319,179.656,6.245,149.231
C04813=1121.959,-6.464,-50.330,179.656,6.249,149.232
C04814=1121.955,-6.248,-50.342,179.657,6.253,149.233
C04815=1121.951,-6.033,-50.353,179.658,6.257,149.233
C04816=1121.946,-5.819,-50.365,179.658,6.260,149.234
C04817=1121.942,-5.603,-50.376,179.658,6.265,149.235
C04818=1121.937,-5.387,-50.387,179.659,6.269,149.235
C04819=1121.932,-5.139,-50.401,179.659,6.273,149.236
C04820=1121.927,-4.889,-50.414,179.660,6.278,149.237
C04821=1121.922,-4.639,-50.427,179.661,6.282,149.238
C04822=1121.917,-4.390,-50.441,179.661,6.287,149.239
C04823=1121.912,-4.140,-50.454,179.662,6.291,149.239
C04824=1121.906,-3.890,-50.467,179.662,6.295,149.240
C04825=1121.902,-3.641,-50.480,179.663,6.300,149.241
C04826=1121.896,-3.391,-50.494,179.664,6.304,149.242
C04827=1121.892,-3.141,-50.507,179.664,6.309,149.243
C04828=1121.886,-2.892,-50.521,179.665,6.314,149.244
C04829=1121.881,-2.642,-50.534,179.666,6.318,149.244
C04830=1121.876,-2.393,-50.547,179.666,6.323,149.245
C04831=1121.870,-2.144,-50.561,179.667,6.328,149.246
C04832=1121.866,-1.894,-50.574,179.667,6.332,149.247
C04833=1121.860,-1.645,-50.587,179.668,6.336,149.248
C04834=1121.855,-1.395,-50.600,179.668,6.341,149.249
C04835=1121.850,-1.145,-50.614,179.669,6.345,149.249
C04836=1121.845,-0.895,-50.628,179.669,6.350,149.250
C04837=1121.840,-0.646,-50.641,179.670,6.354,149.251
C04838=1121.835,-0.396,-50.655,179.671,6.359,149.252
C04839=1121.829,-0.147,-50.667,179.671,6.364,149.253
C04840=1121.825,0.103,-50.682,179.672,6.367,149.253
C04841=1121.819,0.353,-50.695,179.672,6.372,149.254
C04842=1121.814,0.602,-50.709,179.673,6.377,149.255
C04843=1121.809,0.852,-50.722,179.673,6.382,149.256
C04844=1121.804,1.101,-50.736,179.674,6.386,149.257
C04845=1121.799,1.351,-50.749,179.675,6.391,149.258
C04846=1121.794,1.600,-50.763,179.676,6.395,149.258
C04847=1121.788,1.850,-50.776,179.675,6.399,149.259
C04848=1121.783,2.099,-50.790,179.676,6.404,149.260
C04849=1121.778,2.349,-50.803,179.677,6.408,149.261
C04850=1121.773,2.599,-50.818,179.677,6.413,149.262
C04851=1121.768,2.848,-50.831,179.678,6.418,149.263
C04852=1121.763,3.098,-50.844,179.679,6.422,149.264
C04853=1121.758,3.347,-50.858,179.678,6.426,149.264
C04854=1121.753,3.597,-50.871,179.680,6.431,149.265
C04855=1121.748,3.846,-50.885,179.680,6.435,149.266
C04856=1121.743,4.096,-50.900,179.681,6.440,149.267
C04857=1121.738,4.346,-50.913,179.681,6.445,149.268
C04858=1121.732,4.595,-50.926,179.682,6.450,149.269
C04859=1121.728,4.845,-50.941,179.682,6.453,149.269
C04860=1121.722,5.094,-50.954,179.683,6.458,149.270
C04861=1121.717,5.344,-50.968,179.683,6.463,149.271
C04862=1121.712,5.593,-50.982,179.684,6.467,149.272
C04863=1121.707,5.843,-50.995,179.684,6.472,149.273
C04864=1121.702,6.093,-51.009,179.685,6.477,149.274
C04865=1121.697,6.342,-51.024,179.685,6.481,149.275
C04866=1121.692,6.592,-51.036,179.686,6.485,149.275
C04867=1121.687,6.807,-51.049,179.686,6.489,149.276
C04868=1121.683,7.022,-51.061,179.687,6.493,149.277
C04869=1121.679,7.237,-51.073,179.687,6.497,149.278
C04870=1121.674,7.451,-51.085,179.687,6.501,149.278
C04871=1121.670,7.666,-51.096,179.688,6.505,149.279
C04872=1121.665,7.882,-51.109,179.688,6.509,149.280
C04873=1121.661,8.097,-51.120,179.688,6.512,149.281
C04874=1121.656,8.311,-51.132,179.689,6.516,149.281
C04875=1121.652,8.561,-51.147,179.690,6.522,149.282
C04876=1121.646,8.811,-51.160,179.690,6.526,149.283
C04877=1121.641,9.060,-51.174,179.691,6.531,149.284
C04878=1121.636,9.310,-51.188,179.692,6.535,149.284
C04879=1121.632,9.559,-51.202,179.693,6.540,149.285
C04880=1121.627,9.809,-51.216,179.693,6.545,149.286
C04881=1121.621,10.059,-51.229,179.694,6.549,149.287
C04882=1121.616,10.308,-51.244,179.695,6.554,149.288
C04883=1121.611,10.558,-51.258,179.695,6.558,149.289
C04884=1121.605,10.807,-51.272,179.696,6.563,149.289
C04885=1121.600,11.057,-51.286,179.697,6.568,149.290
C04886=1121.595,11.307,-51.300,179.698,6.573,149.291
C04887=1121.590,11.556,-51.315,179.699,6.577,149.292
C04888=1121.585,11.805,-51.329,179.700,6.582,149.293
C04889=1121.580,12.055,-51.343,179.701,6.586,149.293
C04890=1121.576,12.304,-51.357,179.701,6.591,149.294
C04891=1121.570,12.553,-51.371,179.702,6.596,149.295
C04892=1121.565,12.803,-51.385,179.703,6.600,149.296
C04893=1121.560,13.053,-51.398,179.703,6.605,149.297
C04894=1121.555,13.303,-51.413,179.704,6.609,149.297
C04895=1121.550,13.553,-51.427,179.705,6.614,149.298
C04896=1121.544,13.802,-51.441,179.706,6.618,149.299
C04897=1121.539,14.052,-51.455,179.706,6.623,149.300
C04898=1121.535,14.301,-51.469,179.707,6.628,149.300
C04899=1121.530,14.550,-51.484,179.708,6.632,149.301
C04900=1121.524,14.799,-51.498,179.709,6.637,149.302
C04901=1121.519,15.049,-51.513,179.710,6.641,149.303
C04902=1121.514,15.299,-51.527,179.710,6.646,149.304
C04903=1121.509,15.549,-51.541,179.712,6.651,149.304
C04904=1121.504,15.798,-51.555,179.712,6.656,149.305
C04905=1121.499,16.047,-51.569,179.713,6.660,149.306
C04906=1121.493,16.297,-51.584,179.714,6.665,149.307
C04907=1121.488,16.547,-51.598,179.715,6.669,149.307
C04908=1121.483,16.797,-51.613,179.716,6.673,149.308
C04909=1121.478,17.046,-51.627,179.717,6.678,149.309
C04910=1121.474,17.296,-51.642,179.718,6.682,149.309
C04911=1121.468,17.545,-51.656,179.718,6.687,149.310
C04912=1121.463,17.794,-51.670,179.719,6.691,149.311
C04913=1121.458,18.044,-51.684,179.720,6.696,149.312
C04914=1121.453,18.294,-51.699,179.721,6.700,149.313
C04915=1121.448,18.543,-51.713,179.722,6.705,149.313
C04916=1121.444,18.792,-51.728,179.723,6.709,149.314
C04917=1121.438,19.042,-51.743,179.724,6.714,149.315
C04918=1121.433,19.292,-51.757,179.725,6.718,149.315
C04919=1121.428,19.541,-51.771,179.725,6.723,149.316
C04920=1121.423,19.790,-51.786,179.726,6.727,149.317
C04921=1121.418,20.040,-51.800,179.727,6.731,149.318
C04922=1121.413,20.290,-51.815,179.728,6.736,149.318
C04923=1121.408,20.505,-51.828,179.729,6.740,149.319
C04924=1121.404,20.719,-51.840,179.729,6.744,149.320
C04925=1121.400,20.935,-51.852,179.730,6.747,149.320
C04926=1121.395,21.150,-51.865,179.731,6.751,149.321
C04927=1121.391,21.364,-51.878,179.732,6.755,149.321
C04928=1121.386,21.579,-51.891,179.733,6.759,149.322
C04929=1121.383,21.794,-51.903,179.733,6.763,149.323
C04930=1121.378,22.010,-51.915,179.734,6.767,149.323
C04931=1121.373,22.259,-51.930,179.735,6.771,149.324
C04932=1121.368,22.508,-51.945,179.736,6.776,149.325
C04933=1121.363,22.758,-51.960,179.737,6.780,149.325
C04934=1121.358,23.008,-51.974,179.738,6.785,149.326
C04935=1121.352,23.257,-51.988,179.739,6.789,149.327
C04936=1121.348,23.506,-52.003,179.740,6.793,149.328
C04937=1121.343,23.755,-52.018,179.741,6.798,149.328
C04938=1121.337,24.005,-52.033,179.742,6.802,149.329
C04939=1121.332,24.254,-52.048,179.743,6.807,149.330
C04940=1121.327,24.504,-52.062,179.744,6.811,149.330
C04941=1121.322,24.754,-52.077,179.745,6.815,149.331
C04942=1121.317,25.003,-52.092,179.746,6.820,149.332
C04943=1121.312,25.252,-52.107,179.747,6.824,149.332
C04944=1121.307,25.502,-52.122,179.747,6.829,149.333
C04945=1121.302,25.751,-52.137,179.748,6.833,149.334
C04946=1121.297,26.001,-52.151,179.750,6.837,149.335
C04947=1121.292,26.251,-52.166,179.751,6.842,149.335
C04948=1121.287,26.500,-52.181,179.752,6.846,149.336
C04949=1121.282,26.749,-52.196,179.753,6.850,149.336
C04950=1121.276,26.999,-52.211,179.753,6.855,149.337
C04951=1121.272,27.249,-52.226,179.754,6.859,149.338
C04952=1121.267,27.498,-52.240,179.755,6.864,149.339
C04953=1121.261,27.748,-52.255,179.756,6.867,149.339
C04954=1121.257,27.997,-52.270,179.757,6.871,149.340
C04955=1121.252,28.247,-52.286,179.758,6.876,149.341
C04956=1121.247,28.497,-52.301,179.759,6.880,149.341
C04957=1121.242,28.746,-52.315,179.760,6.884,149.342
C04958=1121.237,28.996,-52.330,179.761,6.889,149.343
C04959=1121.232,29.245,-52.345,179.762,6.893,149.343
C04960=1121.226,29.495,-52.360,179.763,6.897,149.344
C04961=1121.222,29.744,-52.375,179.764,6.902,149.344
C04962=1121.216,29.993,-52.391,179.765,6.906,149.345
C04963=1121.211,30.243,-52.405,179.766,6.911,149.346
C04964=1121.207,30.492,-52.420,179.767,6.915,149.347
C04965=1121.201,30.741,-52.436,179.768,6.919,149.347
C04966=1121.196,30.991,-52.450,179.769,6.924,149.348
C04967=1121.191,31.241,-52.466,179.770,6.928,149.349
C04968=1121.187,31.490,-52.481,179.771,6.932,149.349
C04969=1121.181,31.740,-52.497,179.772,6.936,149.350
C04970=1121.177,31.989,-52.511,179.773,6.941,149.351
C04971=1121.171,32.239,-52.526,179.774,6.945,149.351
C04972=1121.166,32.488,-52.541,179.775,6.949,149.352
C04973=1121.161,32.737,-52.557,179.776,6.954,149.353
C04974=1121.156,32.987,-52.571,179.778,6.958,149.353
C04975=1121.151,33.237,-52.587,179.779,6.962,149.354
C04976=1121.146,33.487,-52.603,179.780,6.966,149.354
C04977=1121.141,33.736,-52.618,179.781,6.971,149.355
C04978=1121.136,33.985,-52.633,179.782,6.975,149.356
C04979=1121.131,34.200,-52.646,179.783,6.978,149.356
C04980=1121.127,34.415,-52.659,179.784,6.982,149.357
C04981=1121.123,34.629,-52.673,179.785,6.986,149.357
C04982=1121.119,34.845,-52.686,179.786,6.989,149.358
C04983=1121.115,35.060,-52.699,179.787,6.993,149.358
C04984=1121.110,35.274,-52.713,179.788,6.996,149.359
C04985=1121.106,35.489,-52.726,179.788,7.000,149.359
C04986=1121.101,35.704,-52.739,179.790,7.004,149.360
C04987=1121.096,35.953,-52.754,179.791,7.008,149.361
C04988=1121.091,36.202,-52.769,179.792,7.013,149.361
C04989=1121.086,36.452,-52.785,179.793,7.017,149.362
C04990=1121.082,36.702,-52.800,179.793,7.020,149.362
C04991=1121.076,36.951,-52.816,179.794,7.025,149.363
C04992=1121.071,37.200,-52.831,179.795,7.029,149.364
C04993=1121.067,37.450,-52.847,179.797,7.033,149.364
C04994=1121.061,37.700,-52.862,179.798,7.037,149.365
C04995=1121.056,37.949,-52.878,179.799,7.042,149.366
C04996=1121.051,38.198,-52.893,179.800,7.046,149.366
C04997=1121.046,38.447,-52.908,179.801,7.050,149.367
C04998=1121.041,38.698,-52.924,179.802,7.054,149.367
C04999=1121.037,38.947,-52.939,179.804,7.058,149.368
C05000=1121.031,39.196,-52.955,179.805,7.063,149.369
C05001=1121.026,39.445,-52.971,179.806,7.067,149.369
C05002=1121.021,39.696,-52.986,179.807,7.071,149.370
C05003=1121.016,39.945,-53.001,179.808,7.076,149.370
C05004=1121.011,40.194,-53.017,179.810,7.079,149.371
C05005=1121.006,40.444,-53.033,179.811,7.084,149.372
C05006=1121.001,40.694,-53.049,179.811,7.087,149.372
C05007=1120.996,40.942,-53.064,179.812,7.092,149.373
C05008=1120.991,41.191,-53.080,179.813,7.096,149.374
C05009=1120.986,41.442,-53.096,179.815,7.100,149.374
C05010=1120.981,41.691,-53.111,179.816,7.104,149.375
C05011=1120.976,41.940,-53.126,179.817,7.108,149.375
C05012=1120.971,42.190,-53.142,179.818,7.113,149.376
C05013=1120.966,42.439,-53.159,179.820,7.117,149.376
C05014=1120.961,42.688,-53.174,179.821,7.121,149.377
C05015=1120.956,42.938,-53.190,179.822,7.125,149.378
C05016=1120.952,43.187,-53.205,179.823,7.129,149.378
C05017=1120.946,43.437,-53.221,179.824,7.134,149.379
C05018=1120.942,43.686,-53.237,179.825,7.138,149.379
C05019=1120.936,43.936,-53.253,179.826,7.141,149.380
C05020=1120.931,44.185,-53.269,179.827,7.145,149.380
C05021=1120.926,44.435,-53.285,179.829,7.150,149.381
C05022=1120.921,44.684,-53.301,179.830,7.154,149.382
C05023=1120.916,44.933,-53.316,179.831,7.158,149.382
C05024=1120.912,45.183,-53.332,179.832,7.162,149.383
C05025=1120.907,45.432,-53.348,179.833,7.166,149.383
C05026=1120.902,45.682,-53.364,179.835,7.170,149.384
C05027=1120.896,45.932,-53.380,179.836,7.175,149.385
C05028=1120.891,46.180,-53.396,179.837,7.179,149.385
C05029=1120.886,46.430,-53.412,179.839,7.183,149.386
C05030=1120.881,46.680,-53.428,179.840,7.187,149.386
C05031=1120.877,46.929,-53.444,179.841,7.191,149.387
C05032=1120.871,47.179,-53.460,179.842,7.195,149.387
C05033=1120.866,47.429,-53.476,179.843,7.199,149.388
C05034=1120.861,47.678,-53.492,179.844,7.203,149.388
C05035=1120.857,47.892,-53.506,179.845,7.207,149.389
C05036=1120.853,48.108,-53.519,179.846,7.210,149.389
C05037=1120.849,48.322,-53.533,179.847,7.213,149.390
C05038=1120.844,48.536,-53.547,179.849,7.217,149.390
C05039=1120.841,48.751,-53.561,179.849,7.221,149.391
C05040=1120.836,48.966,-53.575,179.850,7.224,149.391
C05041=1120.831,49.180,-53.589,179.852,7.228,149.392
C05042=1120.828,49.395,-53.603,179.853,7.231,149.392
C05043=1120.822,49.645,-53.618,179.854,7.235,149.393
C05044=1120.818,49.894,-53.635,179.855,7.240,149.394
C05045=1120.812,50.144,-53.651,179.856,7.243,149.394
C05046=1120.808,50.393,-53.667,179.857,7.248,149.395
C05047=1120.803,50.642,-53.683,179.859,7.252,149.395
C05048=1120.798,50.891,-53.699,179.860,7.256,149.396
C05049=1120.793,51.141,-53.715,179.862,7.260,149.396
C05050=1120.788,51.390,-53.731,179.863,7.264,149.397
C05051=1120.783,51.640,-53.747,179.863,7.268,149.397
C05052=1120.778,51.889,-53.764,179.865,7.272,149.398
C05053=1120.772,52.139,-53.780,179.866,7.276,149.399
C05054=1120.767,52.388,-53.796,179.867,7.280,149.399
C05055=1120.763,52.638,-53.813,179.869,7.284,149.400
C05056=1120.758,52.888,-53.829,179.870,7.288,149.400
C05057=1120.753,53.137,-53.845,179.871,7.292,149.401
C05058=1120.748,53.386,-53.862,179.873,7.296,149.401
C05059=1120.743,53.635,-53.878,179.874,7.301,149.402
C05060=1120.739,53.885,-53.894,179.875,7.304,149.402
C05061=1120.733,54.134,-53.911,179.876,7.309,149.403
C05062=1120.728,54.384,-53.927,179.878,7.313,149.403
C05063=1120.723,54.633,-53.943,179.879,7.316,149.404
C05064=1120.718,54.882,-53.960,179.880,7.320,149.404
C05065=1120.713,55.132,-53.976,179.881,7.324,149.405
C05066=1120.708,55.381,-53.992,179.883,7.328,149.405
C05067=1120.703,55.631,-54.010,179.884,7.333,149.406
C05068=1120.698,55.880,-54.026,179.885,7.337,149.406
C05069=1120.693,56.130,-54.042,179.886,7.341,149.407
C05070=1120.688,56.379,-54.058,179.888,7.345,149.408
C05071=1120.684,56.628,-54.075,179.889,7.349,149.408
C05072=1120.679,56.878,-54.092,179.891,7.353,149.409
C05073=1120.673,57.127,-54.108,179.892,7.357,149.409
C05074=1120.669,57.377,-54.124,179.893,7.360,149.410
C05075=1120.664,57.626,-54.141,179.894,7.364,149.410
C05076=1120.658,57.876,-54.158,179.895,7.369,149.411
C05077=1120.654,58.125,-54.175,179.897,7.372,149.411
C05078=1120.649,58.374,-54.191,179.898,7.377,149.412
C05079=1120.644,58.624,-54.208,179.900,7.381,149.412
C05080=1120.639,58.874,-54.224,179.901,7.385,149.413
C05081=1120.634,59.122,-54.240,179.902,7.389,149.413
C05082=1120.629,59.372,-54.257,179.904,7.393,149.414
C05083=1120.624,59.621,-54.274,179.905,7.397,149.414
C05084=1120.619,59.871,-54.291,179.906,7.401,149.415
C05085=1120.615,60.120,-54.307,179.908,7.405,149.416
C05086=1120.609,60.369,-54.324,179.909,7.408,149.416
C05087=1120.604,60.619,-54.341,179.910,7.413,149.417
C05088=1120.600,60.868,-54.358,179.911,7.417,149.417
C05089=1120.595,61.118,-54.375,179.913,7.421,149.417
C05090=1120.589,61.367,-54.391,179.914,7.425,149.418
C05091=1120.585,61.582,-54.406,179.915,7.429,149.419
C05092=1120.581,61.796,-54.420,179.916,7.432,149.419
C05093=1120.577,62.011,-54.435,179.917,7.435,149.419
C05094=1120.572,62.225,-54.449,179.919,7.439,149.420
C05095=1120.568,62.440,-54.464,179.920,7.442,149.420
C05096=1120.564,62.654,-54.478,179.921,7.445,149.421
C05097=1120.559,62.870,-54.492,179.922,7.449,149.421
C05098=1120.555,63.083,-54.507,179.923,7.452,149.422
C05099=1120.550,63.333,-54.524,179.924,7.456,149.422
C05100=1120.546,63.583,-54.541,179.926,7.460,149.423
C05101=1120.541,63.832,-54.557,179.927,7.464,149.423
C05102=1120.535,64.081,-54.574,179.929,7.469,149.424
C05103=1120.531,64.331,-54.591,179.930,7.472,149.424
C05104=1120.526,64.581,-54.608,179.932,7.476,149.425
C05105=1120.522,64.830,-54.626,179.933,7.481,149.425
C05106=1120.516,65.079,-54.643,179.934,7.484,149.426
C05107=1120.511,65.328,-54.659,179.935,7.488,149.426
C05108=1120.506,65.578,-54.677,179.936,7.492,149.427
C05109=1120.502,65.827,-54.693,179.938,7.496,149.427
C05110=1120.496,66.077,-54.710,179.940,7.500,149.428
C05111=1120.492,66.325,-54.727,179.941,7.504,149.428
C05112=1120.486,66.575,-54.745,179.942,7.508,149.429
C05113=1120.482,66.825,-54.761,179.944,7.512,149.429
C05114=1120.477,67.074,-54.779,179.945,7.516,149.430
C05115=1120.472,67.324,-54.795,179.947,7.520,149.430
C05116=1120.467,67.572,-54.813,179.948,7.524,149.431
C05117=1120.462,67.822,-54.830,179.949,7.528,149.431
C05118=1120.457,68.072,-54.847,179.951,7.532,149.432
C05119=1120.453,68.320,-54.864,179.952,7.536,149.432
C05120=1120.448,68.570,-54.882,179.953,7.540,149.433
C05121=1120.442,68.820,-54.899,179.954,7.543,149.433
C05122=1120.437,69.069,-54.915,179.956,7.547,149.434
C05123=1120.432,69.318,-54.933,179.957,7.552,149.434
C05124=1120.428,69.568,-54.950,179.959,7.556,149.435
C05125=1120.423,69.817,-54.968,179.960,7.559,149.435
C05126=1120.418,70.067,-54.985,179.962,7.563,149.436
C05127=1120.413,70.316,-55.002,179.963,7.568,149.436
C05128=1120.408,70.565,-55.020,179.965,7.572,149.437
C05129=1120.403,70.814,-55.037,179.966,7.575,149.437
C05130=1120.398,71.064,-55.053,179.967,7.580,149.438
C05131=1120.393,71.313,-55.071,179.969,7.584,149.438
C05132=1120.389,71.562,-55.088,179.970,7.588,149.439
C05133=1120.384,71.812,-55.106,179.972,7.591,149.439
C05134=1120.379,72.061,-55.123,179.973,7.596,149.440
C05135=1120.374,72.311,-55.141,179.975,7.600,149.440
C05136=1120.369,72.560,-55.158,179.976,7.603,149.440
C05137=1120.364,72.809,-55.176,179.977,7.607,149.441
C05138=1120.359,73.059,-55.193,179.978,7.611,149.442
C05139=1120.354,73.307,-55.210,179.980,7.615,149.442
C05140=1120.349,73.557,-55.227,179.981,7.619,149.442
C05141=1120.344,73.806,-55.245,179.983,7.623,149.443
C05142=1120.339,74.056,-55.263,179.984,7.627,149.443
C05143=1120.335,74.305,-55.280,179.986,7.631,149.444
C05144=1120.330,74.555,-55.297,179.987,7.635,149.444
C05145=1120.325,74.804,-55.315,179.988,7.639,149.445
C05146=1120.319,75.054,-55.332,179.990,7.643,149.445
C05147=1120.316,75.268,-55.347,179.991,7.646,149.446
C05148=1120.312,75.483,-55.363,179.993,7.650,149.446
C05149=1120.307,75.697,-55.378,179.993,7.653,149.447
C05150=1120.303,75.911,-55.393,179.995,7.657,149.447
C05151=1120.299,76.126,-55.408,179.996,7.660,149.448
C05152=1120.294,76.340,-55.423,179.997,7.663,149.448
C05153=1120.291,76.555,-55.438,179.999,7.667,149.448
C05154=1120.287,76.769,-55.454,180.000,7.670,149.449
C05155=1120.281,77.019,-55.471,-179.999,7.674,149.449
C05156=1120.277,77.268,-55.489,-179.998,7.678,149.450
C05157=1120.272,77.517,-55.507,-179.997,7.681,149.450
C05158=1120.266,77.767,-55.524,-179.996,7.685,149.451
C05159=1120.261,78.016,-55.542,-179.995,7.688,149.451
C05160=1120.257,78.265,-55.559,-179.994,7.692,149.452
C05161=1120.252,78.514,-55.577,-179.993,7.696,149.453
C05162=1120.247,78.764,-55.595,-179.992,7.700,149.453
C05163=1120.242,79.013,-55.613,-179.992,7.703,149.454
C05164=1120.237,79.263,-55.631,-179.990,7.707,149.454
C05165=1120.232,79.512,-55.649,-179.990,7.711,149.455
C05166=1120.227,79.762,-55.666,-179.988,7.715,149.455
C05167=1120.222,80.011,-55.684,-179.987,7.718,149.456
C05168=1120.217,80.260,-55.702,-179.986,7.722,149.456
C05169=1120.213,80.509,-55.719,-179.985,7.726,149.457
C05170=1120.208,80.758,-55.737,-179.984,7.729,149.457
C05171=1120.203,81.008,-55.754,-179.983,7.734,149.458
C05172=1120.198,81.257,-55.772,-179.982,7.737,149.459
C05173=1120.194,81.507,-55.791,-179.981,7.741,149.459
C05174=1120.189,81.756,-55.809,-179.980,7.744,149.460
C05175=1120.184,82.005,-55.827,-179.978,7.749,149.460
C05176=1120.179,82.254,-55.845,-179.978,7.752,149.461
C05177=1120.174,82.504,-55.862,-179.976,7.756,149.461
C05178=1120.169,82.753,-55.880,-179.975,7.760,149.462
C05179=1120.164,83.003,-55.898,-179.974,7.763,149.462
C05180=1120.159,83.252,-55.916,-179.973,7.767,149.463
C05181=1120.154,83.501,-55.934,-179.971,7.771,149.463
C05182=1120.149,83.750,-55.952,-179.971,7.775,149.464
C05183=1120.145,84.000,-55.970,-179.969,7.778,149.464
C05184=1120.140,84.249,-55.988,-179.968,7.783,149.465
C05185=1120.135,84.498,-56.006,-179.967,7.786,149.465
C05186=1120.130,84.747,-56.024,-179.965,7.790,149.466
C05187=1120.125,84.997,-56.042,-179.964,7.794,149.466
C05188=1120.121,85.246,-56.060,-179.963,7.797,149.467
C05189=1120.116,85.495,-56.078,-179.962,7.801,149.467
C05190=1120.111,85.745,-56.096,-179.961,7.805,149.468
C05191=1120.106,85.994,-56.114,-179.959,7.809,149.468
C05192=1120.101,86.243,-56.132,-179.958,7.813,149.469
C05193=1120.096,86.493,-56.151,-179.957,7.817,149.469
C05194=1120.091,86.742,-56.169,-179.955,7.821,149.470
C05195=1120.086,86.991,-56.187,-179.954,7.825,149.471
C05196=1120.082,87.241,-56.205,-179.953,7.828,149.471
C05197=1120.077,87.490,-56.223,-179.952,7.832,149.471
C05198=1120.072,87.739,-56.241,-179.950,7.836,149.472
C05199=1120.067,87.988,-56.259,-179.949,7.840,149.473
C05200=1120.062,88.238,-56.277,-179.947,7.844,149.473
C05201=1120.058,88.487,-56.296,-179.946,7.847,149.473
C05202=1120.052,88.736,-56.315,-179.945,7.851,149.474
C05203=1120.048,88.951,-56.330,-179.944,7.854,149.474
C05204=1120.044,89.166,-56.346,-179.942,7.858,149.475
C05205=1120.040,89.379,-56.361,-179.941,7.861,149.475
C05206=1120.036,89.594,-56.377,-179.940,7.864,149.476
C05207=1120.032,89.808,-56.393,-179.939,7.868,149.476
C05208=1120.028,90.023,-56.408,-179.938,7.871,149.476
C05209=1120.023,90.238,-56.424,-179.937,7.874,149.477
C05210=1120.019,90.452,-56.440,-179.935,7.878,149.477
C05211=1120.014,90.701,-56.458,-179.933,7.882,149.478
C05212=1120.009,90.950,-56.476,-179.932,7.885,149.478
C05213=1120.005,91.199,-56.495,-179.931,7.889,149.479
C05214=1119.999,91.449,-56.514,-179.929,7.893,149.479
C05215=1119.995,91.698,-56.532,-179.928,7.897,149.479
C05216=1119.990,91.947,-56.550,-179.927,7.901,149.480
C05217=1119.986,92.197,-56.569,-179.925,7.905,149.480
C05218=1119.980,92.446,-56.587,-179.923,7.909,149.481
C05219=1119.975,92.695,-56.605,-179.922,7.913,149.481
C05220=1119.971,92.945,-56.625,-179.920,7.917,149.482
C05221=1119.966,93.194,-56.643,-179.919,7.920,149.482
C05222=1119.960,93.443,-56.661,-179.917,7.924,149.483
C05223=1119.956,93.692,-56.680,-179.915,7.928,149.483
C05224=1119.952,93.942,-56.698,-179.914,7.932,149.483
C05225=1119.946,94.191,-56.717,-179.912,7.936,149.484
C05226=1119.941,94.440,-56.735,-179.911,7.939,149.484
C05227=1119.937,94.690,-56.754,-179.910,7.943,149.485
C05228=1119.931,94.939,-56.772,-179.908,7.947,149.485
C05229=1119.927,95.188,-56.791,-179.906,7.951,149.486
C05230=1119.922,95.437,-56.809,-179.905,7.955,149.486
C05231=1119.917,95.686,-56.829,-179.903,7.959,149.486
C05232=1119.912,95.935,-56.847,-179.901,7.963,149.487
C05233=1119.908,96.185,-56.866,-179.899,7.967,149.487
C05234=1119.903,96.434,-56.884,-179.898,7.971,149.488
C05235=1119.899,96.683,-56.903,-179.896,7.975,149.488
C05236=1119.893,96.933,-56.922,-179.894,7.978,149.488
C05237=1119.888,97.182,-56.941,-179.892,7.982,149.489
C05238=1119.884,97.431,-56.959,-179.891,7.986,149.489
C05239=1119.879,97.680,-56.978,-179.889,7.990,149.490
C05240=1119.874,97.929,-56.996,-179.888,7.994,149.490
C05241=1119.869,98.179,-57.016,-179.886,7.998,149.491
C05242=1119.864,98.428,-57.034,-179.884,8.001,149.491
C05243=1119.859,98.678,-57.054,-179.882,8.005,149.491
C05244=1119.854,98.927,-57.071,-179.881,8.009,149.492
C05245=1119.850,99.177,-57.091,-179.879,8.013,149.492
C05246=1119.845,99.425,-57.110,-179.878,8.017,149.493
C05247=1119.840,99.674,-57.128,-179.875,8.021,149.493
C05248=1119.835,99.924,-57.147,-179.873,8.025,149.493
C05249=1119.831,100.172,-57.166,-179.872,8.029,149.494
C05250=1119.826,100.423,-57.185,-179.870,8.033,149.494
C05251=1119.820,100.671,-57.204,-179.868,8.036,149.494
C05252=1119.816,100.921,-57.223,-179.866,8.040,149.495
C05253=1119.811,101.170,-57.242,-179.864,8.044,149.495
C05254=1119.807,101.419,-57.261,-179.862,8.048,149.495
C05255=1119.801,101.668,-57.280,-179.861,8.052,149.496
C05256=1119.797,101.917,-57.299,-179.859,8.056,149.496
C05257=1119.792,102.167,-57.318,-179.857,8.060,149.496
C05258=1119.787,102.416,-57.337,-179.855,8.063,149.497
C05259=1119.783,102.631,-57.354,-179.853,8.067,149.497
C05260=1119.779,102.845,-57.370,-179.851,8.071,149.497
C05261=1119.775,103.059,-57.387,-179.850,8.073,149.498
C05262=1119.771,103.273,-57.403,-179.848,8.077,149.498
C05263=1119.766,103.488,-57.419,-179.847,8.080,149.498
C05264=1119.763,103.702,-57.435,-179.845,8.083,149.498
C05265=1119.758,103.916,-57.452,-179.843,8.087,149.499
C05266=1119.754,104.130,-57.468,-179.842,8.090,149.499
C05267=1119.749,104.380,-57.488,-179.840,8.094,149.499
C05268=1119.744,104.629,-57.507,-179.837,8.098,149.500
C05269=1119.740,104.878,-57.526,-179.835,8.102,149.500
C05270=1119.734,105.128,-57.545,-179.834,8.106,149.500
C05271=1119.730,105.377,-57.565,-179.832,8.109,149.501
C05272=1119.726,105.626,-57.584,-179.829,8.113,149.501
C05273=1119.720,105.875,-57.603,-179.827,8.117,149.501
C05274=1119.716,106.125,-57.623,-179.825,8.121,149.501
C05275=1119.710,106.374,-57.642,-179.823,8.124,149.502
C05276=1119.706,106.623,-57.661,-179.821,8.129,149.502
C05277=1119.701,106.872,-57.680,-179.819,8.132,149.502
C05278=1119.696,107.121,-57.700,-179.817,8.136,149.503
C05279=1119.692,107.371,-57.719,-179.814,8.140,149.503
C05280=1119.687,107.619,-57.738,-179.813,8.144,149.503
C05281=1119.682,107.869,-57.758,-179.811,8.148,149.503
C05282=1119.677,108.119,-57.777,-179.808,8.152,149.504
C05283=1119.672,108.367,-57.797,-179.806,8.155,149.504
C05284=1119.668,108.617,-57.816,-179.804,8.159,149.504
C05285=1119.663,108.866,-57.835,-179.802,8.163,149.505
C05286=1119.658,109.115,-57.855,-179.799,8.167,149.505
C05287=1119.653,109.364,-57.875,-179.797,8.171,149.505
C05288=1119.648,109.613,-57.894,-179.795,8.174,149.505
C05289=1119.644,109.862,-57.913,-179.793,8.178,149.505
C05290=1119.639,110.112,-57.933,-179.791,8.182,149.506
C05291=1119.634,110.361,-57.952,-179.789,8.185,149.506
C05292=1119.629,110.610,-57.972,-179.786,8.190,149.506
C05293=1119.625,110.859,-57.992,-179.784,8.193,149.506
C05294=1119.620,111.108,-58.012,-179.782,8.197,149.507
C05295=1119.615,111.358,-58.031,-179.780,8.201,149.507
C05296=1119.610,111.607,-58.051,-179.778,8.204,149.507
C05297=1119.605,111.856,-58.070,-179.776,8.208,149.507
C05298=1119.601,112.105,-58.090,-179.774,8.211,149.508
C05299=1119.596,112.354,-58.110,-179.772,8.215,149.508
C05300=1119.592,112.604,-58.129,-179.770,8.218,149.508
C05301=1119.586,112.852,-58.149,-179.769,8.221,149.509
C05302=1119.582,113.102,-58.169,-179.767,8.225,149.509
C05303=1119.577,113.351,-58.189,-179.765,8.229,149.509
C05304=1119.572,113.600,-58.208,-179.763,8.232,149.509
C05305=1119.567,113.849,-58.228,-179.761,8.236,149.510
C05306=1119.562,114.099,-58.248,-179.759,8.239,149.510
C05307=1119.558,114.348,-58.268,-179.758,8.242,149.510
C05308=1119.553,114.596,-58.288,-179.756,8.246,149.511
C05309=1119.548,114.846,-58.307,-179.754,8.249,149.511
C05310=1119.544,115.095,-58.328,-179.752,8.253,149.511
C05311=1119.539,115.345,-58.347,-179.750,8.256,149.511
C05312=1119.534,115.594,-58.367,-179.748,8.260,149.512
C05313=1119.529,115.842,-58.387,-179.747,8.263,149.512
C05314=1119.524,116.092,-58.407,-179.745,8.267,149.512
C05315=1119.520,116.306,-58.424,-179.744,8.269,149.513
C05316=1119.516,116.521,-58.441,-179.742,8.273,149.513
C05317=1119.512,116.735,-58.459,-179.740,8.276,149.513
C05318=1119.508,116.948,-58.476,-179.739,8.278,149.513
C05319=1119.504,117.163,-58.493,-179.737,8.281,149.513
C05320=1119.500,117.377,-58.510,-179.735,8.284,149.514
C05321=1119.495,117.591,-58.527,-179.734,8.287,149.514
C05322=1119.492,117.806,-58.544,-179.732,8.290,149.514
C05323=1119.487,118.055,-58.565,-179.730,8.293,149.514
C05324=1119.482,118.304,-58.584,-179.729,8.297,149.515
C05325=1119.478,118.553,-58.604,-179.727,8.301,149.515
C05326=1119.472,118.803,-58.625,-179.725,8.303,149.515
C05327=1119.468,119.051,-58.645,-179.723,8.307,149.515
C05328=1119.463,119.301,-58.665,-179.721,8.310,149.516
C05329=1119.459,119.550,-58.685,-179.719,8.314,149.516
C05330=1119.453,119.798,-58.705,-179.718,8.317,149.516
C05331=1119.449,120.048,-58.725,-179.716,8.321,149.517
C05332=1119.444,120.297,-58.745,-179.714,8.324,149.517
C05333=1119.439,120.547,-58.765,-179.712,8.328,149.517
C05334=1119.434,120.796,-58.786,-179.711,8.331,149.517
C05335=1119.430,121.045,-58.806,-179.709,8.334,149.518
C05336=1119.425,121.294,-58.826,-179.707,8.338,149.518
C05337=1119.421,121.543,-58.846,-179.705,8.341,149.518
C05338=1119.416,121.792,-58.867,-179.704,8.344,149.518
C05339=1119.410,122.041,-58.886,-179.701,8.348,149.519
C05340=1119.406,122.290,-58.907,-179.699,8.351,149.519
C05341=1119.401,122.539,-58.927,-179.698,8.354,149.519
C05342=1119.397,122.788,-58.948,-179.696,8.358,149.520
C05343=1119.391,123.038,-58.968,-179.694,8.361,149.520
C05344=1119.387,123.287,-58.988,-179.692,8.365,149.520
C05345=1119.383,123.536,-59.009,-179.691,8.368,149.520
C05346=1119.378,123.785,-59.029,-179.689,8.371,149.521
C05347=1119.373,124.034,-59.050,-179.687,8.375,149.521
C05348=1119.368,124.284,-59.070,-179.686,8.378,149.521
C05349=1119.364,124.533,-59.090,-179.684,8.381,149.521
C05350=1119.359,124.781,-59.110,-179.682,8.385,149.522
C05351=1119.354,125.031,-59.131,-179.680,8.389,149.522
C05352=1119.350,125.280,-59.152,-179.678,8.391,149.522
C05353=1119.345,125.529,-59.172,-179.676,8.395,149.523
C05354=1119.340,125.779,-59.192,-179.674,8.398,149.523
C05355=1119.335,126.027,-59.213,-179.673,8.401,149.523
C05356=1119.331,126.276,-59.233,-179.671,8.405,149.523
C05357=1119.326,126.526,-59.254,-179.669,8.408,149.524
C05358=1119.321,126.775,-59.274,-179.668,8.411,149.524
C05359=1119.317,127.024,-59.295,-179.666,8.415,149.524
C05360=1119.312,127.273,-59.316,-179.664,8.418,149.525
C05361=1119.307,127.522,-59.336,-179.663,8.421,149.525
C05362=1119.302,127.771,-59.357,-179.661,8.425,149.525
C05363=1119.298,128.020,-59.377,-179.659,8.428,149.525
C05364=1119.293,128.269,-59.398,-179.657,8.431,149.526
C05365=1119.288,128.518,-59.419,-179.655,8.435,149.526
C05366=1119.284,128.767,-59.439,-179.653,8.438,149.526
C05367=1119.278,129.016,-59.460,-179.652,8.441,149.527
C05368=1119.274,129.265,-59.480,-179.650,8.445,149.527
C05369=1119.269,129.515,-59.501,-179.648,8.448,149.527
C05370=1119.264,129.764,-59.522,-179.647,8.451,149.527
C05371=1119.261,129.978,-59.540,-179.645,8.454,149.527
C05372=1119.257,130.192,-59.557,-179.644,8.458,149.528
C05373=1119.252,130.407,-59.575,-179.642,8.460,149.528
C05374=1119.248,130.620,-59.593,-179.641,8.463,149.528
C05375=1119.244,130.835,-59.610,-179.639,8.466,149.529
C05376=1119.240,131.048,-59.629,-179.638,8.468,149.529
C05377=1119.236,131.263,-59.647,-179.636,8.471,149.529
C05378=1119.232,131.477,-59.664,-179.635,8.474,149.529
C05379=1119.227,131.726,-59.685,-179.633,8.477,149.529
C05380=1119.222,131.975,-59.706,-179.631,8.481,149.530
C05381=1119.218,132.224,-59.726,-179.630,8.484,149.530
C05382=1119.213,132.473,-59.748,-179.628,8.487,149.530
C05383=1119.209,132.722,-59.769,-179.626,8.491,149.531
C05384=1119.204,132.971,-59.789,-179.625,8.494,149.531
C05385=1119.199,133.221,-59.810,-179.623,8.498,149.531
C05386=1119.194,133.470,-59.831,-179.622,8.501,149.532
C05387=1119.189,133.718,-59.852,-179.620,8.504,149.532
C05388=1119.185,133.967,-59.873,-179.618,8.508,149.532
C05389=1119.180,134.216,-59.894,-179.617,8.511,149.533
C05390=1119.176,134.466,-59.915,-179.614,8.514,149.533
C05391=1119.171,134.715,-59.936,-179.612,8.518,149.533
C05392=1119.166,134.964,-59.957,-179.611,8.521,149.533
C05393=1119.161,135.213,-59.978,-179.609,8.524,149.534
C05394=1119.156,135.462,-59.999,-179.608,8.527,149.534
C05395=1119.152,135.711,-60.020,-179.606,8.531,149.534
C05396=1119.147,135.961,-60.041,-179.604,8.534,149.535
C05397=1119.142,136.210,-60.062,-179.603,8.537,149.535
C05398=1119.138,136.458,-60.083,-179.601,8.541,149.535
C05399=1119.133,136.707,-60.104,-179.600,8.544,149.535
C05400=1119.128,136.957,-60.125,-179.598,8.547,149.536
C05401=1119.124,137.205,-60.146,-179.596,8.551,149.536
C05402=1119.119,137.455,-60.167,-179.594,8.554,149.536
C05403=1119.114,137.704,-60.188,-179.593,8.558,149.537
C05404=1119.110,137.953,-60.209,-179.591,8.561,149.537
C05405=1119.105,138.202,-60.230,-179.589,8.564,149.537
C05406=1119.100,138.451,-60.252,-179.588,8.568,149.538
C05407=1119.096,138.700,-60.273,-179.586,8.570,149.538
C05408=1119.091,138.949,-60.295,-179.585,8.574,149.538
C05409=1119.086,139.198,-60.315,-179.583,8.578,149.539
C05410=1119.081,139.447,-60.336,-179.581,8.581,149.539
C05411=1119.077,139.696,-60.358,-179.579,8.584,149.539
C05412=1119.072,139.946,-60.379,-179.578,8.587,149.539
C05413=1119.067,140.194,-60.401,-179.576,8.591,149.540
C05414=1119.063,140.443,-60.421,-179.575,8.594,149.540
C05415=1119.058,140.692,-60.443,-179.573,8.597,149.541
C05416=1119.053,140.941,-60.465,-179.571,8.601,149.541
C05417=1119.048,141.190,-60.486,-179.570,8.604,149.541
C05418=1119.044,141.440,-60.508,-179.568,8.608,149.541
C05419=1119.040,141.689,-60.528,-179.567,8.611,149.542
C05420=1119.035,141.937,-60.550,-179.565,8.614,149.542
C05421=1119.030,142.187,-60.571,-179.563,8.618,149.543
C05422=1119.025,142.436,-60.593,-179.562,8.621,149.543
C05423=1119.020,142.685,-60.614,-179.560,8.625,149.543
C05424=1119.016,142.933,-60.635,-179.559,8.627,149.543
C05425=1119.012,143.183,-60.657,-179.557,8.631,149.544
C05426=1119.007,143.432,-60.678,-179.555,8.635,149.544
C05427=1119.002,143.646,-60.697,-179.554,8.638,149.545
C05428=1118.999,143.859,-60.715,-179.553,8.640,149.545
C05429=1118.994,144.074,-60.733,-179.551,8.643,149.545
C05430=1118.991,144.288,-60.752,-179.550,8.646,149.545
C05431=1118.987,144.502,-60.771,-179.549,8.649,149.546
C05432=1118.982,144.716,-60.788,-179.547,8.652,149.546
C05433=1118.978,144.930,-60.807,-179.546,8.655,149.546
C05434=1118.975,145.144,-60.826,-179.545,8.657,149.547
C05435=1118.970,145.393,-60.847,-179.542,8.662,149.547
C05436=1118.965,145.642,-60.869,-179.540,8.665,149.547
C05437=1118.961,145.891,-60.891,-179.538,8.669,149.547
C05438=1118.956,146.140,-60.912,-179.535,8.673,149.547
C05439=1118.951,146.389,-60.933,-179.533,8.676,149.548
C05440=1118.946,146.639,-60.955,-179.530,8.681,149.548
C05441=1118.942,146.887,-60.977,-179.528,8.684,149.548
C05442=1118.937,147.137,-60.999,-179.526,8.688,149.548
C05443=1118.932,147.385,-61.021,-179.524,8.692,149.549
C05444=1118.928,147.634,-61.042,-179.522,8.695,149.549
C05445=1118.923,147.884,-61.064,-179.519,8.699,149.549
C05446=1118.918,148.132,-61.085,-179.517,8.703,149.549
C05447=1118.914,148.382,-61.108,-179.515,8.707,149.550
C05448=1118.909,148.630,-61.129,-179.513,8.710,149.550
C05449=1118.904,148.879,-61.151,-179.509,8.714,149.550
C05450=1118.900,149.128,-61.173,-179.507,8.718,149.550
C05451=1118.895,149.377,-61.195,-179.505,8.721,149.550
C05452=1118.891,149.626,-61.217,-179.503,8.725,149.551
C05453=1118.886,149.875,-61.238,-179.500,8.729,149.551
C05454=1118.882,150.124,-61.260,-179.498,8.732,149.551
C05455=1118.877,150.373,-61.282,-179.496,8.735,149.551
C05456=1118.872,150.622,-61.304,-179.494,8.739,149.551
C05457=1118.868,150.871,-61.326,-179.491,8.743,149.552
C05458=1118.862,151.120,-61.348,-179.489,8.747,149.552
C05459=1118.858,151.369,-61.370,-179.486,8.750,149.552
C05460=1118.853,151.618,-61.392,-179.484,8.753,149.552
C05461=1118.849,151.867,-61.414,-179.482,8.757,149.552
C05462=1118.844,152.116,-61.436,-179.480,8.761,149.553
C05463=1118.839,152.365,-61.458,-179.477,8.764,149.553
C05464=1118.835,152.614,-61.479,-179.475,8.768,149.553
C05465=1118.830,152.864,-61.502,-179.473,8.771,149.553
C05466=1118.825,153.112,-61.524,-179.470,8.774,149.553
C05467=1118.820,153.362,-61.546,-179.468,8.778,149.553
C05468=1118.816,153.610,-61.568,-179.466,8.782,149.554
C05469=1118.812,153.859,-61.590,-179.463,8.785,149.554
C05470=1118.807,154.109,-61.613,-179.461,8.789,149.554
C05471=1118.802,154.357,-61.634,-179.459,8.792,149.554
C05472=1118.797,154.607,-61.656,-179.456,8.795,149.554
C05473=1118.793,154.855,-61.679,-179.454,8.799,149.554
C05474=1118.789,155.104,-61.701,-179.452,8.802,149.554
C05475=1118.784,155.337,-61.722,-179.450,8.805,149.555
C05476=1118.779,155.571,-61.743,-179.448,8.809,149.555
C05477=1118.775,155.805,-61.764,-179.445,8.812,149.555
C05478=1118.771,156.038,-61.785,-179.443,8.815,149.555
C05479=1118.766,156.272,-61.805,-179.440,8.818,149.555
C05480=1118.762,156.506,-61.827,-179.439,8.821,149.555
C05481=1118.758,156.739,-61.847,-179.437,8.824,149.555
C05482=1118.753,156.973,-61.868,-179.434,8.828,149.556
C05483=1118.750,157.202,-61.889,-179.432,8.831,149.556
C05484=1118.745,157.432,-61.909,-179.430,8.834,149.556
C05485=1118.741,157.661,-61.930,-179.428,8.837,149.556
C05486=1118.736,157.890,-61.950,-179.426,8.840,149.556
